LIN {X -173.235,Y +1142.221,Z +0.000,A -20.000,E1 +22.930,E3 +126000.532,E4 +0.000} C_DIS
LIN {X -181.123,Y +1133.734,Z +0.000,A -20.000,E1 +30.868,E3 +126021.288,E4 +0.000} C_DIS
LIN {X -189.654,Y +1120.856,Z +0.000,A -20.000,E1 +39.018,E3 +126043.302,E4 +0.000} C_DIS
LIN {X -195.246,Y +1107.046,Z +0.000,A -20.000,E1 +44.515,E3 +126061.204,E4 +0.000} C_DIS
LIN {X -198.051,Y +1092.368,Z +0.000,A -20.000,E1 +47.947,E3 +126077.730,E4 +0.000} C_DIS
LIN {X -198.143,Y +1081.370,Z +0.000,A -19.806,E1 +49.153,E3 +126089.591,E4 +0.000} C_DIS
LIN {X -197.177,Y +1073.569,Z +0.000,A -17.356,E1 +49.162,E3 +126098.175,E4 +0.000} C_DIS
LIN {X -195.448,Y +1066.139,Z +0.000,A -12.154,E1 +48.512,E3 +126106.770,E4 +0.000} C_DIS
LIN {X -193.346,Y +1058.941,Z +0.000,A -7.133,E1 +47.724,E3 +126115.650,E4 +0.000} C_DIS
LIN {X -191.781,Y +1050.839,Z +0.000,A -3.715,E1 +47.274,E3 +126125.983,E4 +0.000} C_DIS
LIN {X -190.795,Y +1039.355,Z +0.000,A -0.983,E1 +46.842,E3 +126140.643,E4 +0.000} C_DIS
LIN {X -190.395,Y +1028.856,Z +0.000,A -0.089,E1 +46.598,E3 +126154.037,E4 +0.000} C_DIS
LIN {X -190.239,Y +1018.851,Z +0.000,A -0.004,E1 +46.529,E3 +126166.805,E4 +0.000} C_DIS
LIN {X -190.161,Y +1004.975,Z +0.000,A +0.000,E1 +46.506,E3 +126184.519,E4 +0.000} C_DIS
LIN {X -190.142,Y +412.853,Z +0.000,A +0.000,E1 +46.501,E3 +126940.725,E4 +0.000} C_DIS
LIN {X -190.147,Y +401.077,Z +0.000,A +0.000,E1 +46.499,E3 +126955.766,E4 +0.000} C_DIS
LIN {X -190.159,Y +390.929,Z +0.000,A +0.000,E1 +46.494,E3 +126968.732,E4 +0.000} C_DIS
LIN {X -190.174,Y +383.973,Z +0.000,A +0.000,E1 +46.484,E3 +126977.625,E4 +0.000} C_DIS
LIN {X -190.200,Y +373.815,Z +0.000,A +0.000,E1 +46.448,E3 +126990.630,E4 +0.000} C_DIS
LIN {X -190.154,Y +361.003,Z +0.000,A +0.000,E1 +46.303,E3 +127007.124,E4 +0.000} C_DIS
LIN {X -189.772,Y +350.660,Z +0.000,A +0.049,E1 +45.996,E3 +127020.663,E4 +0.000} C_DIS
LIN {X -189.325,Y +346.917,Z +0.000,A +0.243,E1 +45.771,E3 +127025.732,E4 +0.000} C_DIS
LIN {X -188.196,Y +342.754,Z +0.000,A +1.966,E1 +45.249,E3 +127031.740,E4 +0.000} C_DIS
LIN {X -185.199,Y +337.023,Z +0.000,A +6.630,E1 +43.793,E3 +127041.114,E4 +0.000} C_DIS
LIN {X -181.141,Y +331.596,Z +0.000,A +12.274,E1 +41.569,E3 +127051.674,E4 +0.000} C_DIS
LIN {X -176.762,Y +326.804,Z +0.000,A +17.560,E1 +38.898,E3 +127063.098,E4 +0.000} C_DIS
LIN {X -172.184,Y +322.578,Z +0.000,A +19.859,E1 +36.197,E3 +127075.828,E4 +0.000} C_DIS
LIN {X -165.998,Y +317.874,Z +0.000,A +20.000,E1 +32.027,E3 +127095.586,E4 +0.000} C_DIS
LIN {X -160.137,Y +314.334,Z +0.000,A +20.000,E1 +26.368,E3 +127119.955,E4 +0.000} C_DIS
LIN {X -155.624,Y +312.245,Z +0.000,A +20.000,E1 +19.506,E3 +127148.631,E4 +0.000} C_DIS
LIN {X -153.557,Y +311.879,Z +0.000,A +20.000,E1 +11.113,E3 +127184.386,E4 +0.000} C_DIS
LIN {X -155.320,Y +313.348,Z +0.000,A +20.000,E1 +3.401,E3 +127217.570,E4 +0.000} C_DIS
LIN {X -160.005,Y +315.804,Z +0.000,A +20.000,E1 -4.720,E3 +127247.948,E4 +0.000} C_DIS
LIN {X -164.504,Y +318.255,Z +0.000,A +20.000,E1 -10.663,E3 +127267.317,E4 +0.000} C_DIS
LIN {X -170.340,Y +322.684,Z +0.000,A +20.000,E1 -17.457,E3 +127287.349,E4 +0.000} C_DIS
LIN {X -175.568,Y +329.106,Z +0.000,A +20.000,E1 -24.747,E3 +127304.583,E4 +0.000} C_DIS
LIN {X -184.074,Y +340.065,Z +0.000,A +20.000,E1 -33.664,E3 +127327.523,E4 +0.000} C_DIS
LIN {X -190.779,Y +351.388,Z +0.000,A +20.000,E1 -40.083,E3 +127345.301,E4 +0.000} C_DIS
LIN {X -195.254,Y +362.955,Z +0.000,A +20.000,E1 -44.515,E3 +127360.054,E4 +0.000} C_DIS
LIN {X -197.754,Y +374.780,Z +0.000,A +20.000,E1 -47.450,E3 +127373.476,E4 +0.000} C_DIS
LIN {X -198.310,Y +383.215,Z +0.000,A +19.956,E1 -48.698,E3 +127382.600,E4 +0.000} C_DIS
LIN {X -197.912,Y +391.275,Z +0.000,A +18.601,E1 -49.158,E3 +127391.318,E4 +0.000} C_DIS
LIN {X -196.679,Y +398.944,Z +0.000,A +13.989,E1 -48.784,E3 +127399.872,E4 +0.000} C_DIS
LIN {X -194.742,Y +406.288,Z +0.000,A +8.476,E1 -48.001,E3 +127408.555,E4 +0.000} C_DIS
LIN {X -192.748,Y +413.472,Z +0.000,A +3.905,E1 -47.267,E3 +127417.565,E4 +0.000} C_DIS
LIN {X -191.781,Y +419.162,Z +0.000,A +1.739,E1 -46.975,E3 +127424.833,E4 +0.000} C_DIS
LIN {X -190.795,Y +430.646,Z +0.000,A +0.152,E1 -46.707,E3 +127439.494,E4 +0.000} C_DIS
LIN {X -190.395,Y +441.145,Z +0.000,A +0.001,E1 -46.583,E3 +127452.887,E4 +0.000} C_DIS
LIN {X -190.239,Y +451.150,Z +0.000,A -0.000,E1 -46.528,E3 +127465.655,E4 +0.000} C_DIS
LIN {X -190.161,Y +465.026,Z +0.000,A -0.000,E1 -46.506,E3 +127483.370,E4 +0.000} C_DIS
LIN {X -190.142,Y +1057.148,Z +0.000,A -0.000,E1 -46.500,E3 +128239.576,E4 +0.000} C_DIS
LIN {X -190.147,Y +1068.924,Z +0.000,A -0.000,E1 -46.499,E3 +128254.617,E4 +0.000} C_DIS
LIN {X -190.159,Y +1079.072,Z +0.000,A -0.000,E1 -46.493,E3 +128267.582,E4 +0.000} C_DIS
LIN {X -190.174,Y +1086.028,Z +0.000,A -0.000,E1 -46.483,E3 +128276.476,E4 +0.000} C_DIS
LIN {X -190.200,Y +1096.186,Z +0.000,A -0.000,E1 -46.448,E3 +128289.480,E4 +0.000} C_DIS
LIN {X -190.154,Y +1108.998,Z +0.000,A -0.054,E1 -46.295,E3 +128305.975,E4 +0.000} C_DIS
LIN {X -189.772,Y +1119.341,Z +0.000,A -0.752,E1 -45.902,E3 +128319.513,E4 +0.000} C_DIS
LIN {X -189.097,Y +1124.276,Z +0.000,A -2.508,E1 -45.397,E3 +128326.245,E4 +0.000} C_DIS
LIN {X -187.410,Y +1129.069,Z +0.000,A -5.304,E1 -44.585,E3 +128333.418,E4 +0.000} C_DIS
LIN {X -183.899,Y +1134.873,Z +0.000,A -10.372,E1 -42.805,E3 +128343.424,E4 +0.000} C_DIS
LIN {X -179.711,Y +1140.065,Z +0.000,A -15.940,E1 -40.393,E3 +128354.210,E4 +0.000} C_DIS
LIN {X -176.763,Y +1143.197,Z +0.000,A -18.748,E1 -38.674,E3 +128361.948,E4 +0.000} C_DIS
LIN {X -172.185,Y +1147.423,Z +0.000,A -19.971,E1 -36.175,E3 +128374.678,E4 +0.000} C_DIS
LIN {X -165.999,Y +1152.127,Z +0.000,A -20.000,E1 -32.027,E3 +128394.436,E4 +0.000} C_DIS
LIN {X -160.138,Y +1155.667,Z +0.000,A -20.000,E1 -26.368,E3 +128418.806,E4 +0.000} C_DIS
LIN {X -155.625,Y +1157.756,Z +0.000,A -20.000,E1 -19.505,E3 +128447.482,E4 +0.000} C_DIS
LIN {X -153.552,Y +1158.113,Z +0.000,A -20.000,E1 -11.113,E3 +128483.233,E4 +0.000} C_DIS
LIN {X -156.311,Y +1155.540,Z +0.000,A -20.000,E1 -0.839,E3 +128526.593,E4 +0.000} C_DIS
LIN {X -161.281,Y +1151.851,Z +0.000,A -20.000,E1 +7.737,E3 +128556.492,E4 +0.000} C_DIS
LIN {X -167.493,Y +1147.157,Z +0.000,A -20.000,E1 +16.195,E3 +128580.931,E4 +0.000} C_DIS
LIN {X -173.235,Y +1142.221,Z +0.000,A -20.000,E1 +22.930,E3 +128598.233,E4 +0.000} C_DIS
LIN {X -181.123,Y +1133.734,Z +0.000,A -20.000,E1 +30.868,E3 +128618.989,E4 +0.000} C_DIS
LIN {X -189.654,Y +1120.856,Z +0.000,A -20.000,E1 +39.018,E3 +128641.003,E4 +0.000} C_DIS
LIN {X -195.246,Y +1107.046,Z +0.000,A -20.000,E1 +44.515,E3 +128658.905,E4 +0.000} C_DIS
LIN {X -198.051,Y +1092.368,Z +0.000,A -20.000,E1 +47.947,E3 +128675.431,E4 +0.000} C_DIS
LIN {X -198.143,Y +1081.370,Z +0.000,A -19.806,E1 +49.153,E3 +128687.292,E4 +0.000} C_DIS
LIN {X -197.177,Y +1073.569,Z +0.000,A -17.356,E1 +49.162,E3 +128695.876,E4 +0.000} C_DIS
LIN {X -195.448,Y +1066.139,Z +0.000,A -12.154,E1 +48.512,E3 +128704.471,E4 +0.000} C_DIS
LIN {X -193.346,Y +1058.941,Z +0.000,A -7.133,E1 +47.724,E3 +128713.351,E4 +0.000} C_DIS
LIN {X -191.781,Y +1050.839,Z +0.000,A -3.715,E1 +47.274,E3 +128723.684,E4 +0.000} C_DIS
LIN {X -190.795,Y +1039.355,Z +0.000,A -0.983,E1 +46.842,E3 +128738.344,E4 +0.000} C_DIS
LIN {X -190.395,Y +1028.856,Z +0.000,A -0.089,E1 +46.598,E3 +128751.738,E4 +0.000} C_DIS
LIN {X -190.239,Y +1018.851,Z +0.000,A -0.004,E1 +46.529,E3 +128764.506,E4 +0.000} C_DIS
LIN {X -190.161,Y +1004.975,Z +0.000,A +0.000,E1 +46.506,E3 +128782.220,E4 +0.000} C_DIS
LIN {X -190.142,Y +412.853,Z +0.000,A +0.000,E1 +46.501,E3 +129538.426,E4 +0.000} C_DIS
LIN {X -190.147,Y +401.077,Z +0.000,A +0.000,E1 +46.499,E3 +129553.467,E4 +0.000} C_DIS
LIN {X -190.159,Y +390.929,Z +0.000,A +0.000,E1 +46.494,E3 +129566.433,E4 +0.000} C_DIS
LIN {X -190.174,Y +383.973,Z +0.000,A +0.000,E1 +46.484,E3 +129575.326,E4 +0.000} C_DIS
LIN {X -190.200,Y +373.815,Z +0.000,A +0.000,E1 +46.448,E3 +129588.331,E4 +0.000} C_DIS
LIN {X -190.154,Y +361.003,Z +0.000,A +0.000,E1 +46.303,E3 +129604.825,E4 +0.000} C_DIS
LIN {X -189.772,Y +350.660,Z +0.000,A +0.049,E1 +45.996,E3 +129618.364,E4 +0.000} C_DIS
LIN {X -189.325,Y +346.917,Z +0.000,A +0.243,E1 +45.771,E3 +129623.433,E4 +0.000} C_DIS
LIN {X -188.196,Y +342.754,Z +0.000,A +1.966,E1 +45.249,E3 +129629.441,E4 +0.000} C_DIS
LIN {X -185.199,Y +337.023,Z +0.000,A +6.630,E1 +43.793,E3 +129638.815,E4 +0.000} C_DIS
LIN {X -181.141,Y +331.596,Z +0.000,A +12.274,E1 +41.569,E3 +129649.375,E4 +0.000} C_DIS
LIN {X -176.762,Y +326.804,Z +0.000,A +17.560,E1 +38.898,E3 +129660.799,E4 +0.000} C_DIS
LIN {X -172.184,Y +322.578,Z +0.000,A +19.859,E1 +36.197,E3 +129673.529,E4 +0.000} C_DIS
LIN {X -165.998,Y +317.874,Z +0.000,A +20.000,E1 +32.027,E3 +129693.287,E4 +0.000} C_DIS
LIN {X -160.137,Y +314.334,Z +0.000,A +20.000,E1 +26.368,E3 +129717.656,E4 +0.000} C_DIS
LIN {X -155.624,Y +312.245,Z +0.000,A +20.000,E1 +19.506,E3 +129746.332,E4 +0.000} C_DIS
LIN {X -153.557,Y +311.879,Z +0.000,A +20.000,E1 +11.113,E3 +129782.087,E4 +0.000} C_DIS
LIN {X -155.320,Y +313.348,Z +0.000,A +20.000,E1 +3.401,E3 +129815.271,E4 +0.000} C_DIS
LIN {X -160.005,Y +315.804,Z +0.000,A +20.000,E1 -4.720,E3 +129845.649,E4 +0.000} C_DIS
LIN {X -164.504,Y +318.255,Z +0.000,A +20.000,E1 -10.663,E3 +129865.018,E4 +0.000} C_DIS
LIN {X -170.340,Y +322.684,Z +0.000,A +20.000,E1 -17.457,E3 +129885.050,E4 +0.000} C_DIS
LIN {X -175.568,Y +329.106,Z +0.000,A +20.000,E1 -24.747,E3 +129902.284,E4 +0.000} C_DIS
LIN {X -184.074,Y +340.065,Z +0.000,A +20.000,E1 -33.664,E3 +129925.224,E4 +0.000} C_DIS
LIN {X -190.779,Y +351.388,Z +0.000,A +20.000,E1 -40.083,E3 +129943.002,E4 +0.000} C_DIS
LIN {X -195.254,Y +362.955,Z +0.000,A +20.000,E1 -44.515,E3 +129957.755,E4 +0.000} C_DIS
LIN {X -197.754,Y +374.780,Z +0.000,A +20.000,E1 -47.450,E3 +129971.177,E4 +0.000} C_DIS
LIN {X -198.310,Y +383.215,Z +0.000,A +19.956,E1 -48.698,E3 +129980.301,E4 +0.000} C_DIS
LIN {X -197.912,Y +391.275,Z +0.000,A +18.601,E1 -49.158,E3 +129989.019,E4 +0.000} C_DIS
LIN {X -196.679,Y +398.944,Z +0.000,A +13.989,E1 -48.784,E3 +129997.573,E4 +0.000} C_DIS
LIN {X -194.742,Y +406.288,Z +0.000,A +8.476,E1 -48.001,E3 +130006.256,E4 +0.000} C_DIS
LIN {X -192.748,Y +413.472,Z +0.000,A +3.905,E1 -47.267,E3 +130015.266,E4 +0.000} C_DIS
LIN {X -191.781,Y +419.162,Z +0.000,A +1.739,E1 -46.975,E3 +130022.534,E4 +0.000} C_DIS
LIN {X -190.795,Y +430.646,Z +0.000,A +0.152,E1 -46.707,E3 +130037.195,E4 +0.000} C_DIS
LIN {X -190.395,Y +441.145,Z +0.000,A +0.001,E1 -46.583,E3 +130050.588,E4 +0.000} C_DIS
LIN {X -190.239,Y +451.150,Z +0.000,A -0.000,E1 -46.528,E3 +130063.356,E4 +0.000} C_DIS
LIN {X -190.161,Y +465.026,Z +0.000,A -0.000,E1 -46.506,E3 +130081.071,E4 +0.000} C_DIS
LIN {X -190.142,Y +1057.148,Z +0.000,A -0.000,E1 -46.500,E3 +130837.277,E4 +0.000} C_DIS
LIN {X -190.147,Y +1068.924,Z +0.000,A -0.000,E1 -46.499,E3 +130852.318,E4 +0.000} C_DIS
LIN {X -190.159,Y +1079.072,Z +0.000,A -0.000,E1 -46.493,E3 +130865.283,E4 +0.000} C_DIS
LIN {X -190.174,Y +1086.028,Z +0.000,A -0.000,E1 -46.483,E3 +130874.177,E4 +0.000} C_DIS
LIN {X -190.200,Y +1096.186,Z +0.000,A -0.000,E1 -46.448,E3 +130887.181,E4 +0.000} C_DIS
LIN {X -190.154,Y +1108.998,Z +0.000,A -0.054,E1 -46.295,E3 +130903.676,E4 +0.000} C_DIS
LIN {X -189.772,Y +1119.341,Z +0.000,A -0.752,E1 -45.902,E3 +130917.214,E4 +0.000} C_DIS
LIN {X -189.097,Y +1124.276,Z +0.000,A -2.508,E1 -45.397,E3 +130923.946,E4 +0.000} C_DIS
LIN {X -187.410,Y +1129.069,Z +0.000,A -5.304,E1 -44.585,E3 +130931.119,E4 +0.000} C_DIS
LIN {X -183.899,Y +1134.873,Z +0.000,A -10.372,E1 -42.805,E3 +130941.125,E4 +0.000} C_DIS
LIN {X -179.711,Y +1140.065,Z +0.000,A -15.940,E1 -40.393,E3 +130951.911,E4 +0.000} C_DIS
LIN {X -176.763,Y +1143.197,Z +0.000,A -18.748,E1 -38.674,E3 +130959.649,E4 +0.000} C_DIS
LIN {X -172.185,Y +1147.423,Z +0.000,A -19.971,E1 -36.175,E3 +130972.379,E4 +0.000} C_DIS
LIN {X -165.999,Y +1152.127,Z +0.000,A -20.000,E1 -32.027,E3 +130992.137,E4 +0.000} C_DIS
LIN {X -160.138,Y +1155.667,Z +0.000,A -20.000,E1 -26.368,E3 +131016.507,E4 +0.000} C_DIS
LIN {X -155.625,Y +1157.756,Z +0.000,A -20.000,E1 -19.505,E3 +131045.183,E4 +0.000} C_DIS
LIN {X -153.552,Y +1158.113,Z +0.000,A -20.000,E1 -11.113,E3 +131080.934,E4 +0.000} C_DIS
LIN {X -156.311,Y +1155.540,Z +0.000,A -20.000,E1 -0.839,E3 +131124.294,E4 +0.000} C_DIS
LIN {X -161.281,Y +1151.851,Z +0.000,A -20.000,E1 +7.737,E3 +131154.193,E4 +0.000} C_DIS
LIN {X -167.493,Y +1147.157,Z +0.000,A -20.000,E1 +16.195,E3 +131178.632,E4 +0.000} C_DIS
LIN {X -173.235,Y +1142.221,Z +0.000,A -20.000,E1 +22.930,E3 +131195.934,E4 +0.000} C_DIS
LIN {X -181.123,Y +1133.734,Z +0.000,A -20.000,E1 +30.868,E3 +131216.690,E4 +0.000} C_DIS
LIN {X -189.654,Y +1120.856,Z +0.000,A -20.000,E1 +39.018,E3 +131238.704,E4 +0.000} C_DIS
LIN {X -195.246,Y +1107.046,Z +0.000,A -20.000,E1 +44.515,E3 +131256.606,E4 +0.000} C_DIS
LIN {X -198.051,Y +1092.368,Z +0.000,A -20.000,E1 +47.947,E3 +131273.132,E4 +0.000} C_DIS
LIN {X -198.143,Y +1081.370,Z +0.000,A -19.806,E1 +49.153,E3 +131284.993,E4 +0.000} C_DIS
LIN {X -197.177,Y +1073.569,Z +0.000,A -17.356,E1 +49.162,E3 +131293.577,E4 +0.000} C_DIS
LIN {X -195.448,Y +1066.139,Z +0.000,A -12.154,E1 +48.512,E3 +131302.172,E4 +0.000} C_DIS
LIN {X -193.346,Y +1058.941,Z +0.000,A -7.133,E1 +47.724,E3 +131311.052,E4 +0.000} C_DIS
LIN {X -191.781,Y +1050.839,Z +0.000,A -3.715,E1 +47.274,E3 +131321.385,E4 +0.000} C_DIS
LIN {X -190.795,Y +1039.355,Z +0.000,A -0.983,E1 +46.842,E3 +131336.045,E4 +0.000} C_DIS
LIN {X -190.395,Y +1028.856,Z +0.000,A -0.089,E1 +46.598,E3 +131349.439,E4 +0.000} C_DIS
LIN {X -190.239,Y +1018.851,Z +0.000,A -0.004,E1 +46.529,E3 +131362.207,E4 +0.000} C_DIS
LIN {X -190.161,Y +1004.975,Z +0.000,A +0.000,E1 +46.506,E3 +131379.921,E4 +0.000} C_DIS
LIN {X -190.142,Y +412.853,Z +0.000,A +0.000,E1 +46.501,E3 +132136.127,E4 +0.000} C_DIS
LIN {X -190.147,Y +401.077,Z +0.000,A +0.000,E1 +46.499,E3 +132151.168,E4 +0.000} C_DIS
LIN {X -190.159,Y +390.929,Z +0.000,A +0.000,E1 +46.494,E3 +132164.134,E4 +0.000} C_DIS
LIN {X -190.174,Y +383.973,Z +0.000,A +0.000,E1 +46.484,E3 +132173.027,E4 +0.000} C_DIS
LIN {X -190.200,Y +373.815,Z +0.000,A +0.000,E1 +46.448,E3 +132186.032,E4 +0.000} C_DIS
LIN {X -190.154,Y +361.003,Z +0.000,A +0.000,E1 +46.303,E3 +132202.526,E4 +0.000} C_DIS
LIN {X -189.772,Y +350.660,Z +0.000,A +0.049,E1 +45.996,E3 +132216.065,E4 +0.000} C_DIS
LIN {X -189.325,Y +346.917,Z +0.000,A +0.243,E1 +45.771,E3 +132221.134,E4 +0.000} C_DIS
LIN {X -188.196,Y +342.754,Z +0.000,A +1.966,E1 +45.249,E3 +132227.142,E4 +0.000} C_DIS
LIN {X -185.199,Y +337.023,Z +0.000,A +6.630,E1 +43.793,E3 +132236.516,E4 +0.000} C_DIS
LIN {X -181.141,Y +331.596,Z +0.000,A +12.274,E1 +41.569,E3 +132247.076,E4 +0.000} C_DIS
LIN {X -176.762,Y +326.804,Z +0.000,A +17.560,E1 +38.898,E3 +132258.500,E4 +0.000} C_DIS
LIN {X -172.184,Y +322.578,Z +0.000,A +19.859,E1 +36.197,E3 +132271.230,E4 +0.000} C_DIS
LIN {X -165.998,Y +317.874,Z +0.000,A +20.000,E1 +32.027,E3 +132290.988,E4 +0.000} C_DIS
LIN {X -160.137,Y +314.334,Z +0.000,A +20.000,E1 +26.368,E3 +132315.357,E4 +0.000} C_DIS
LIN {X -155.624,Y +312.245,Z +0.000,A +20.000,E1 +19.506,E3 +132344.033,E4 +0.000} C_DIS
LIN {X -153.557,Y +311.879,Z +0.000,A +20.000,E1 +11.113,E3 +132379.788,E4 +0.000} C_DIS
LIN {X -155.320,Y +313.348,Z +0.000,A +20.000,E1 +3.401,E3 +132412.972,E4 +0.000} C_DIS
LIN {X -160.005,Y +315.804,Z +0.000,A +20.000,E1 -4.720,E3 +132443.350,E4 +0.000} C_DIS
LIN {X -164.504,Y +318.255,Z +0.000,A +20.000,E1 -10.663,E3 +132462.719,E4 +0.000} C_DIS
LIN {X -170.340,Y +322.684,Z +0.000,A +20.000,E1 -17.457,E3 +132482.751,E4 +0.000} C_DIS
LIN {X -175.568,Y +329.106,Z +0.000,A +20.000,E1 -24.747,E3 +132499.985,E4 +0.000} C_DIS
LIN {X -184.074,Y +340.065,Z +0.000,A +20.000,E1 -33.664,E3 +132522.925,E4 +0.000} C_DIS
LIN {X -190.779,Y +351.388,Z +0.000,A +20.000,E1 -40.083,E3 +132540.703,E4 +0.000} C_DIS
LIN {X -195.254,Y +362.955,Z +0.000,A +20.000,E1 -44.515,E3 +132555.456,E4 +0.000} C_DIS
LIN {X -197.754,Y +374.780,Z +0.000,A +20.000,E1 -47.450,E3 +132568.878,E4 +0.000} C_DIS
LIN {X -198.310,Y +383.215,Z +0.000,A +19.956,E1 -48.698,E3 +132578.002,E4 +0.000} C_DIS
LIN {X -197.912,Y +391.275,Z +0.000,A +18.601,E1 -49.158,E3 +132586.720,E4 +0.000} C_DIS
LIN {X -196.679,Y +398.944,Z +0.000,A +13.989,E1 -48.784,E3 +132595.274,E4 +0.000} C_DIS
LIN {X -194.742,Y +406.288,Z +0.000,A +8.476,E1 -48.001,E3 +132603.957,E4 +0.000} C_DIS
LIN {X -192.748,Y +413.472,Z +0.000,A +3.905,E1 -47.267,E3 +132612.967,E4 +0.000} C_DIS
LIN {X -191.781,Y +419.162,Z +0.000,A +1.739,E1 -46.975,E3 +132620.235,E4 +0.000} C_DIS
LIN {X -190.795,Y +430.646,Z +0.000,A +0.152,E1 -46.707,E3 +132634.896,E4 +0.000} C_DIS
LIN {X -190.395,Y +441.145,Z +0.000,A +0.001,E1 -46.583,E3 +132648.289,E4 +0.000} C_DIS
LIN {X -190.239,Y +451.150,Z +0.000,A -0.000,E1 -46.528,E3 +132661.057,E4 +0.000} C_DIS
LIN {X -190.161,Y +465.026,Z +0.000,A -0.000,E1 -46.506,E3 +132678.772,E4 +0.000} C_DIS
LIN {X -190.142,Y +1057.148,Z +0.000,A -0.000,E1 -46.500,E3 +133434.978,E4 +0.000} C_DIS
LIN {X -190.147,Y +1068.924,Z +0.000,A -0.000,E1 -46.499,E3 +133450.019,E4 +0.000} C_DIS
LIN {X -190.159,Y +1079.072,Z +0.000,A -0.000,E1 -46.493,E3 +133462.984,E4 +0.000} C_DIS
LIN {X -190.174,Y +1086.028,Z +0.000,A -0.000,E1 -46.483,E3 +133471.878,E4 +0.000} C_DIS
LIN {X -190.200,Y +1096.186,Z +0.000,A -0.000,E1 -46.448,E3 +133484.882,E4 +0.000} C_DIS
LIN {X -190.154,Y +1108.998,Z +0.000,A -0.054,E1 -46.295,E3 +133501.377,E4 +0.000} C_DIS
LIN {X -189.772,Y +1119.341,Z +0.000,A -0.752,E1 -45.902,E3 +133514.915,E4 +0.000} C_DIS
LIN {X -189.097,Y +1124.276,Z +0.000,A -2.508,E1 -45.397,E3 +133521.647,E4 +0.000} C_DIS
LIN {X -187.410,Y +1129.069,Z +0.000,A -5.304,E1 -44.585,E3 +133528.820,E4 +0.000} C_DIS
LIN {X -183.899,Y +1134.873,Z +0.000,A -10.372,E1 -42.805,E3 +133538.826,E4 +0.000} C_DIS
LIN {X -179.711,Y +1140.065,Z +0.000,A -15.940,E1 -40.393,E3 +133549.612,E4 +0.000} C_DIS
LIN {X -176.763,Y +1143.197,Z +0.000,A -18.748,E1 -38.674,E3 +133557.350,E4 +0.000} C_DIS
LIN {X -172.185,Y +1147.423,Z +0.000,A -19.971,E1 -36.175,E3 +133570.080,E4 +0.000} C_DIS
LIN {X -165.999,Y +1152.127,Z +0.000,A -20.000,E1 -32.027,E3 +133589.838,E4 +0.000} C_DIS
LIN {X -160.138,Y +1155.667,Z +0.000,A -20.000,E1 -26.368,E3 +133614.208,E4 +0.000} C_DIS
LIN {X -155.625,Y +1157.756,Z +0.000,A -20.000,E1 -19.505,E3 +133642.884,E4 +0.000} C_DIS
LIN {X -153.552,Y +1158.113,Z +0.000,A -20.000,E1 -11.113,E3 +133678.635,E4 +0.000} C_DIS
LIN {X -156.311,Y +1155.540,Z +0.000,A -20.000,E1 -0.839,E3 +133721.995,E4 +0.000} C_DIS
LIN {X -161.281,Y +1151.851,Z +0.000,A -20.000,E1 +7.737,E3 +133751.894,E4 +0.000} C_DIS
LIN {X -167.493,Y +1147.157,Z +0.000,A -20.000,E1 +16.195,E3 +133776.333,E4 +0.000} C_DIS
LIN {X -173.235,Y +1142.221,Z +0.000,A -20.000,E1 +22.930,E3 +133793.635,E4 +0.000} C_DIS
LIN {X -181.123,Y +1133.734,Z +0.000,A -20.000,E1 +30.868,E3 +133814.391,E4 +0.000} C_DIS
LIN {X -189.654,Y +1120.856,Z +0.000,A -20.000,E1 +39.018,E3 +133836.405,E4 +0.000} C_DIS
LIN {X -195.246,Y +1107.046,Z +0.000,A -20.000,E1 +44.515,E3 +133854.307,E4 +0.000} C_DIS
LIN {X -198.051,Y +1092.368,Z +0.000,A -20.000,E1 +47.947,E3 +133870.833,E4 +0.000} C_DIS
LIN {X -198.143,Y +1081.370,Z +0.000,A -19.806,E1 +49.153,E3 +133882.694,E4 +0.000} C_DIS
LIN {X -197.177,Y +1073.569,Z +0.000,A -17.356,E1 +49.162,E3 +133891.278,E4 +0.000} C_DIS
LIN {X -195.448,Y +1066.139,Z +0.000,A -12.154,E1 +48.512,E3 +133899.873,E4 +0.000} C_DIS
LIN {X -193.346,Y +1058.941,Z +0.000,A -7.133,E1 +47.724,E3 +133908.753,E4 +0.000} C_DIS
LIN {X -191.781,Y +1050.839,Z +0.000,A -3.715,E1 +47.274,E3 +133919.086,E4 +0.000} C_DIS
LIN {X -190.795,Y +1039.355,Z +0.000,A -0.983,E1 +46.842,E3 +133933.746,E4 +0.000} C_DIS
LIN {X -190.395,Y +1028.856,Z +0.000,A -0.089,E1 +46.598,E3 +133947.140,E4 +0.000} C_DIS
LIN {X -190.239,Y +1018.851,Z +0.000,A -0.004,E1 +46.529,E3 +133959.908,E4 +0.000} C_DIS
LIN {X -190.161,Y +1004.975,Z +0.000,A +0.000,E1 +46.506,E3 +133977.622,E4 +0.000} C_DIS
LIN {X -190.142,Y +412.853,Z +0.000,A +0.000,E1 +46.501,E3 +134733.828,E4 +0.000} C_DIS
LIN {X -190.147,Y +401.077,Z +0.000,A +0.000,E1 +46.499,E3 +134748.869,E4 +0.000} C_DIS
LIN {X -190.159,Y +390.929,Z +0.000,A +0.000,E1 +46.494,E3 +134761.835,E4 +0.000} C_DIS
LIN {X -190.174,Y +383.973,Z +0.000,A +0.000,E1 +46.484,E3 +134770.728,E4 +0.000} C_DIS
LIN {X -190.200,Y +373.815,Z +0.000,A +0.000,E1 +46.448,E3 +134783.733,E4 +0.000} C_DIS
LIN {X -190.154,Y +361.003,Z +0.000,A +0.000,E1 +46.303,E3 +134800.227,E4 +0.000} C_DIS
LIN {X -189.772,Y +350.660,Z +0.000,A +0.049,E1 +45.996,E3 +134813.766,E4 +0.000} C_DIS
LIN {X -189.325,Y +346.917,Z +0.000,A +0.243,E1 +45.771,E3 +134818.835,E4 +0.000} C_DIS
LIN {X -188.196,Y +342.754,Z +0.000,A +1.966,E1 +45.249,E3 +134824.843,E4 +0.000} C_DIS
LIN {X -185.199,Y +337.023,Z +0.000,A +6.630,E1 +43.793,E3 +134834.217,E4 +0.000} C_DIS
LIN {X -181.141,Y +331.596,Z +0.000,A +12.274,E1 +41.569,E3 +134844.777,E4 +0.000} C_DIS
LIN {X -176.762,Y +326.804,Z +0.000,A +17.560,E1 +38.898,E3 +134856.201,E4 +0.000} C_DIS
LIN {X -172.184,Y +322.578,Z +0.000,A +19.859,E1 +36.197,E3 +134868.931,E4 +0.000} C_DIS
LIN {X -165.998,Y +317.874,Z +0.000,A +20.000,E1 +32.027,E3 +134888.689,E4 +0.000} C_DIS
LIN {X -160.137,Y +314.334,Z +0.000,A +20.000,E1 +26.368,E3 +134913.058,E4 +0.000} C_DIS
LIN {X -155.624,Y +312.245,Z +0.000,A +20.000,E1 +19.506,E3 +134941.734,E4 +0.000} C_DIS
LIN {X -153.557,Y +311.879,Z +0.000,A +20.000,E1 +11.113,E3 +134977.489,E4 +0.000} C_DIS
LIN {X -155.320,Y +313.348,Z +0.000,A +20.000,E1 +3.401,E3 +135010.673,E4 +0.000} C_DIS
LIN {X -160.005,Y +315.804,Z +0.000,A +20.000,E1 -4.720,E3 +135041.051,E4 +0.000} C_DIS
LIN {X -164.504,Y +318.255,Z +0.000,A +20.000,E1 -10.663,E3 +135060.420,E4 +0.000} C_DIS
LIN {X -170.340,Y +322.684,Z +0.000,A +20.000,E1 -17.457,E3 +135080.452,E4 +0.000} C_DIS
LIN {X -175.568,Y +329.106,Z +0.000,A +20.000,E1 -24.747,E3 +135097.686,E4 +0.000} C_DIS
LIN {X -184.074,Y +340.065,Z +0.000,A +20.000,E1 -33.664,E3 +135120.626,E4 +0.000} C_DIS
LIN {X -190.779,Y +351.388,Z +0.000,A +20.000,E1 -40.083,E3 +135138.404,E4 +0.000} C_DIS
LIN {X -195.254,Y +362.955,Z +0.000,A +20.000,E1 -44.515,E3 +135153.157,E4 +0.000} C_DIS
LIN {X -197.754,Y +374.780,Z +0.000,A +20.000,E1 -47.450,E3 +135166.579,E4 +0.000} C_DIS
LIN {X -198.310,Y +383.215,Z +0.000,A +19.956,E1 -48.698,E3 +135175.703,E4 +0.000} C_DIS
LIN {X -197.912,Y +391.275,Z +0.000,A +18.601,E1 -49.158,E3 +135184.421,E4 +0.000} C_DIS
LIN {X -196.679,Y +398.944,Z +0.000,A +13.989,E1 -48.784,E3 +135192.975,E4 +0.000} C_DIS
LIN {X -194.742,Y +406.288,Z +0.000,A +8.476,E1 -48.001,E3 +135201.658,E4 +0.000} C_DIS
LIN {X -192.748,Y +413.472,Z +0.000,A +3.905,E1 -47.267,E3 +135210.668,E4 +0.000} C_DIS
LIN {X -191.781,Y +419.162,Z +0.000,A +1.739,E1 -46.975,E3 +135217.936,E4 +0.000} C_DIS
LIN {X -190.795,Y +430.646,Z +0.000,A +0.152,E1 -46.707,E3 +135232.597,E4 +0.000} C_DIS
LIN {X -190.395,Y +441.145,Z +0.000,A +0.001,E1 -46.583,E3 +135245.990,E4 +0.000} C_DIS
LIN {X -190.239,Y +451.150,Z +0.000,A -0.000,E1 -46.528,E3 +135258.758,E4 +0.000} C_DIS
LIN {X -190.161,Y +465.026,Z +0.000,A -0.000,E1 -46.506,E3 +135276.473,E4 +0.000} C_DIS
LIN {X -190.142,Y +1057.148,Z +0.000,A -0.000,E1 -46.500,E3 +136032.679,E4 +0.000} C_DIS
LIN {X -190.147,Y +1068.924,Z +0.000,A -0.000,E1 -46.499,E3 +136047.720,E4 +0.000} C_DIS
LIN {X -190.159,Y +1079.072,Z +0.000,A -0.000,E1 -46.493,E3 +136060.685,E4 +0.000} C_DIS
LIN {X -190.174,Y +1086.028,Z +0.000,A -0.000,E1 -46.483,E3 +136069.579,E4 +0.000} C_DIS
LIN {X -190.200,Y +1096.186,Z +0.000,A -0.000,E1 -46.448,E3 +136082.583,E4 +0.000} C_DIS
LIN {X -190.154,Y +1108.998,Z +0.000,A -0.054,E1 -46.295,E3 +136099.078,E4 +0.000} C_DIS
LIN {X -189.772,Y +1119.341,Z +0.000,A -0.752,E1 -45.902,E3 +136112.616,E4 +0.000} C_DIS
LIN {X -189.097,Y +1124.276,Z +0.000,A -2.508,E1 -45.397,E3 +136119.348,E4 +0.000} C_DIS
LIN {X -187.410,Y +1129.069,Z +0.000,A -5.304,E1 -44.585,E3 +136126.521,E4 +0.000} C_DIS
LIN {X -183.899,Y +1134.873,Z +0.000,A -10.372,E1 -42.805,E3 +136136.527,E4 +0.000} C_DIS
LIN {X -179.711,Y +1140.065,Z +0.000,A -15.940,E1 -40.393,E3 +136147.313,E4 +0.000} C_DIS
LIN {X -176.763,Y +1143.197,Z +0.000,A -18.748,E1 -38.674,E3 +136155.051,E4 +0.000} C_DIS
LIN {X -172.185,Y +1147.423,Z +0.000,A -19.971,E1 -36.175,E3 +136167.781,E4 +0.000} C_DIS
LIN {X -165.999,Y +1152.127,Z +0.000,A -20.000,E1 -32.027,E3 +136187.539,E4 +0.000} C_DIS
LIN {X -160.138,Y +1155.667,Z +0.000,A -20.000,E1 -26.368,E3 +136211.909,E4 +0.000} C_DIS
LIN {X -155.625,Y +1157.756,Z +0.000,A -20.000,E1 -19.505,E3 +136240.585,E4 +0.000} C_DIS
LIN {X -153.552,Y +1158.113,Z +0.000,A -20.000,E1 -11.113,E3 +136276.336,E4 +0.000} C_DIS
LIN {X -156.311,Y +1155.540,Z +0.000,A -20.000,E1 -0.839,E3 +136319.696,E4 +0.000} C_DIS
LIN {X -161.281,Y +1151.851,Z +0.000,A -20.000,E1 +7.737,E3 +136349.595,E4 +0.000} C_DIS
LIN {X -167.493,Y +1147.157,Z +0.000,A -20.000,E1 +16.195,E3 +136374.034,E4 +0.000} C_DIS
LIN {X -173.235,Y +1142.221,Z +0.000,A -20.000,E1 +22.930,E3 +136391.336,E4 +0.000} C_DIS
LIN {X -181.123,Y +1133.734,Z +0.000,A -20.000,E1 +30.868,E3 +136412.092,E4 +0.000} C_DIS
LIN {X -189.654,Y +1120.856,Z +0.000,A -20.000,E1 +39.018,E3 +136434.106,E4 +0.000} C_DIS
LIN {X -195.246,Y +1107.046,Z +0.000,A -20.000,E1 +44.515,E3 +136452.008,E4 +0.000} C_DIS
LIN {X -198.051,Y +1092.368,Z +0.000,A -20.000,E1 +47.947,E3 +136468.534,E4 +0.000} C_DIS
LIN {X -198.143,Y +1081.370,Z +0.000,A -19.806,E1 +49.153,E3 +136480.395,E4 +0.000} C_DIS
LIN {X -197.177,Y +1073.569,Z +0.000,A -17.356,E1 +49.162,E3 +136488.979,E4 +0.000} C_DIS
LIN {X -195.448,Y +1066.139,Z +0.000,A -12.154,E1 +48.512,E3 +136497.574,E4 +0.000} C_DIS
LIN {X -193.346,Y +1058.941,Z +0.000,A -7.133,E1 +47.724,E3 +136506.454,E4 +0.000} C_DIS
LIN {X -191.781,Y +1050.839,Z +0.000,A -3.715,E1 +47.274,E3 +136516.787,E4 +0.000} C_DIS
LIN {X -190.795,Y +1039.355,Z +0.000,A -0.983,E1 +46.842,E3 +136531.447,E4 +0.000} C_DIS
LIN {X -190.395,Y +1028.856,Z +0.000,A -0.089,E1 +46.598,E3 +136544.841,E4 +0.000} C_DIS
LIN {X -190.239,Y +1018.851,Z +0.000,A -0.004,E1 +46.529,E3 +136557.609,E4 +0.000} C_DIS
LIN {X -190.161,Y +1004.975,Z +0.000,A +0.000,E1 +46.506,E3 +136575.323,E4 +0.000} C_DIS
LIN {X -190.142,Y +412.853,Z +0.000,A +0.000,E1 +46.501,E3 +137331.529,E4 +0.000} C_DIS
LIN {X -190.147,Y +401.077,Z +0.000,A +0.000,E1 +46.499,E3 +137346.570,E4 +0.000} C_DIS
LIN {X -190.159,Y +390.929,Z +0.000,A +0.000,E1 +46.494,E3 +137359.536,E4 +0.000} C_DIS
LIN {X -190.174,Y +383.973,Z +0.000,A +0.000,E1 +46.484,E3 +137368.429,E4 +0.000} C_DIS
LIN {X -190.200,Y +373.815,Z +0.000,A +0.000,E1 +46.448,E3 +137381.434,E4 +0.000} C_DIS
LIN {X -190.154,Y +361.003,Z +0.000,A +0.000,E1 +46.303,E3 +137397.928,E4 +0.000} C_DIS
LIN {X -189.772,Y +350.660,Z +0.000,A +0.049,E1 +45.996,E3 +137411.467,E4 +0.000} C_DIS
LIN {X -189.325,Y +346.917,Z +0.000,A +0.243,E1 +45.771,E3 +137416.536,E4 +0.000} C_DIS
LIN {X -188.196,Y +342.754,Z +0.000,A +1.966,E1 +45.249,E3 +137422.544,E4 +0.000} C_DIS
LIN {X -185.199,Y +337.023,Z +0.000,A +6.630,E1 +43.793,E3 +137431.918,E4 +0.000} C_DIS
LIN {X -181.141,Y +331.596,Z +0.000,A +12.274,E1 +41.569,E3 +137442.478,E4 +0.000} C_DIS
LIN {X -176.762,Y +326.804,Z +0.000,A +17.560,E1 +38.898,E3 +137453.902,E4 +0.000} C_DIS
LIN {X -172.184,Y +322.578,Z +0.000,A +19.859,E1 +36.197,E3 +137466.632,E4 +0.000} C_DIS
LIN {X -165.998,Y +317.874,Z +0.000,A +20.000,E1 +32.027,E3 +137486.390,E4 +0.000} C_DIS
LIN {X -160.137,Y +314.334,Z +0.000,A +20.000,E1 +26.368,E3 +137510.759,E4 +0.000} C_DIS
LIN {X -155.624,Y +312.245,Z +0.000,A +20.000,E1 +19.506,E3 +137539.435,E4 +0.000} C_DIS
LIN {X -153.557,Y +311.879,Z +0.000,A +20.000,E1 +11.113,E3 +137575.190,E4 +0.000} C_DIS
LIN {X -155.320,Y +313.348,Z +0.000,A +20.000,E1 +3.401,E3 +137608.374,E4 +0.000} C_DIS
LIN {X -160.005,Y +315.804,Z +0.000,A +20.000,E1 -4.720,E3 +137638.752,E4 +0.000} C_DIS
LIN {X -164.504,Y +318.255,Z +0.000,A +20.000,E1 -10.663,E3 +137658.121,E4 +0.000} C_DIS
LIN {X -170.340,Y +322.684,Z +0.000,A +20.000,E1 -17.457,E3 +137678.153,E4 +0.000} C_DIS
LIN {X -175.568,Y +329.106,Z +0.000,A +20.000,E1 -24.747,E3 +137695.387,E4 +0.000} C_DIS
LIN {X -184.074,Y +340.065,Z +0.000,A +20.000,E1 -33.664,E3 +137718.327,E4 +0.000} C_DIS
LIN {X -190.779,Y +351.388,Z +0.000,A +20.000,E1 -40.083,E3 +137736.105,E4 +0.000} C_DIS
LIN {X -195.254,Y +362.955,Z +0.000,A +20.000,E1 -44.515,E3 +137750.858,E4 +0.000} C_DIS
LIN {X -197.754,Y +374.780,Z +0.000,A +20.000,E1 -47.450,E3 +137764.280,E4 +0.000} C_DIS
LIN {X -198.310,Y +383.215,Z +0.000,A +19.956,E1 -48.698,E3 +137773.404,E4 +0.000} C_DIS
LIN {X -197.912,Y +391.275,Z +0.000,A +18.601,E1 -49.158,E3 +137782.122,E4 +0.000} C_DIS
LIN {X -196.679,Y +398.944,Z +0.000,A +13.989,E1 -48.784,E3 +137790.676,E4 +0.000} C_DIS
LIN {X -194.742,Y +406.288,Z +0.000,A +8.476,E1 -48.001,E3 +137799.359,E4 +0.000} C_DIS
LIN {X -192.748,Y +413.472,Z +0.000,A +3.905,E1 -47.267,E3 +137808.369,E4 +0.000} C_DIS
LIN {X -191.781,Y +419.162,Z +0.000,A +1.739,E1 -46.975,E3 +137815.637,E4 +0.000} C_DIS
LIN {X -190.795,Y +430.646,Z +0.000,A +0.152,E1 -46.707,E3 +137830.298,E4 +0.000} C_DIS
LIN {X -190.395,Y +441.145,Z +0.000,A +0.001,E1 -46.583,E3 +137843.691,E4 +0.000} C_DIS
LIN {X -190.239,Y +451.150,Z +0.000,A -0.000,E1 -46.528,E3 +137856.459,E4 +0.000} C_DIS
LIN {X -190.161,Y +465.026,Z +0.000,A -0.000,E1 -46.506,E3 +137874.174,E4 +0.000} C_DIS
LIN {X -190.142,Y +1057.148,Z +0.000,A -0.000,E1 -46.500,E3 +138630.380,E4 +0.000} C_DIS
LIN {X -190.147,Y +1068.924,Z +0.000,A -0.000,E1 -46.499,E3 +138645.421,E4 +0.000} C_DIS
LIN {X -190.159,Y +1079.072,Z +0.000,A -0.000,E1 -46.493,E3 +138658.386,E4 +0.000} C_DIS
LIN {X -190.174,Y +1086.028,Z +0.000,A -0.000,E1 -46.483,E3 +138667.280,E4 +0.000} C_DIS
LIN {X -190.200,Y +1096.186,Z +0.000,A -0.000,E1 -46.448,E3 +138680.284,E4 +0.000} C_DIS
LIN {X -190.154,Y +1108.998,Z +0.000,A -0.054,E1 -46.295,E3 +138696.779,E4 +0.000} C_DIS
LIN {X -189.772,Y +1119.341,Z +0.000,A -0.752,E1 -45.902,E3 +138710.317,E4 +0.000} C_DIS
LIN {X -189.097,Y +1124.276,Z +0.000,A -2.508,E1 -45.397,E3 +138717.049,E4 +0.000} C_DIS
LIN {X -187.410,Y +1129.069,Z +0.000,A -5.304,E1 -44.585,E3 +138724.222,E4 +0.000} C_DIS
LIN {X -183.899,Y +1134.873,Z +0.000,A -10.372,E1 -42.805,E3 +138734.228,E4 +0.000} C_DIS
LIN {X -179.711,Y +1140.065,Z +0.000,A -15.940,E1 -40.393,E3 +138745.014,E4 +0.000} C_DIS
LIN {X -176.763,Y +1143.197,Z +0.000,A -18.748,E1 -38.674,E3 +138752.752,E4 +0.000} C_DIS
LIN {X -172.185,Y +1147.423,Z +0.000,A -19.971,E1 -36.175,E3 +138765.482,E4 +0.000} C_DIS
LIN {X -165.999,Y +1152.127,Z +0.000,A -20.000,E1 -32.027,E3 +138785.240,E4 +0.000} C_DIS
LIN {X -160.138,Y +1155.667,Z +0.000,A -20.000,E1 -26.368,E3 +138809.610,E4 +0.000} C_DIS
LIN {X -155.625,Y +1157.756,Z +0.000,A -20.000,E1 -19.505,E3 +138838.286,E4 +0.000} C_DIS
LIN {X -153.552,Y +1158.113,Z +0.000,A -20.000,E1 -11.113,E3 +138874.037,E4 +0.000} C_DIS
LIN {X -156.311,Y +1155.540,Z +0.000,A -20.000,E1 -0.839,E3 +138917.397,E4 +0.000} C_DIS
LIN {X -161.281,Y +1151.851,Z +0.000,A -20.000,E1 +7.737,E3 +138947.296,E4 +0.000} C_DIS
LIN {X -167.493,Y +1147.157,Z +0.000,A -20.000,E1 +16.195,E3 +138971.735,E4 +0.000} C_DIS
LIN {X -173.235,Y +1142.221,Z +0.000,A -20.000,E1 +22.930,E3 +138989.037,E4 +0.000} C_DIS
LIN {X -181.123,Y +1133.734,Z +0.000,A -20.000,E1 +30.868,E3 +139009.793,E4 +0.000} C_DIS
LIN {X -189.654,Y +1120.856,Z +0.000,A -20.000,E1 +39.018,E3 +139031.807,E4 +0.000} C_DIS
LIN {X -195.246,Y +1107.046,Z +0.000,A -20.000,E1 +44.515,E3 +139049.709,E4 +0.000} C_DIS
LIN {X -198.051,Y +1092.368,Z +0.000,A -20.000,E1 +47.947,E3 +139066.235,E4 +0.000} C_DIS
LIN {X -198.143,Y +1081.370,Z +0.000,A -19.806,E1 +49.153,E3 +139078.096,E4 +0.000} C_DIS
LIN {X -197.177,Y +1073.569,Z +0.000,A -17.356,E1 +49.162,E3 +139086.680,E4 +0.000} C_DIS
LIN {X -195.448,Y +1066.139,Z +0.000,A -12.154,E1 +48.512,E3 +139095.275,E4 +0.000} C_DIS
LIN {X -193.346,Y +1058.941,Z +0.000,A -7.133,E1 +47.724,E3 +139104.155,E4 +0.000} C_DIS
LIN {X -191.781,Y +1050.839,Z +0.000,A -3.715,E1 +47.274,E3 +139114.488,E4 +0.000} C_DIS
LIN {X -190.795,Y +1039.355,Z +0.000,A -0.983,E1 +46.842,E3 +139129.148,E4 +0.000} C_DIS
LIN {X -190.395,Y +1028.856,Z +0.000,A -0.089,E1 +46.598,E3 +139142.542,E4 +0.000} C_DIS
LIN {X -190.239,Y +1018.851,Z +0.000,A -0.004,E1 +46.529,E3 +139155.310,E4 +0.000} C_DIS
LIN {X -190.161,Y +1004.975,Z +0.000,A +0.000,E1 +46.506,E3 +139173.024,E4 +0.000} C_DIS
LIN {X -190.142,Y +412.853,Z +0.000,A +0.000,E1 +46.501,E3 +139929.230,E4 +0.000} C_DIS
LIN {X -190.147,Y +401.077,Z +0.000,A +0.000,E1 +46.499,E3 +139944.271,E4 +0.000} C_DIS
LIN {X -190.159,Y +390.929,Z +0.000,A +0.000,E1 +46.494,E3 +139957.237,E4 +0.000} C_DIS
LIN {X -190.174,Y +383.973,Z +0.000,A +0.000,E1 +46.484,E3 +139966.130,E4 +0.000} C_DIS
LIN {X -190.200,Y +373.815,Z +0.000,A +0.000,E1 +46.448,E3 +139979.135,E4 +0.000} C_DIS
LIN {X -190.154,Y +361.003,Z +0.000,A +0.000,E1 +46.303,E3 +139995.629,E4 +0.000} C_DIS
LIN {X -189.772,Y +350.660,Z +0.000,A +0.049,E1 +45.996,E3 +140009.168,E4 +0.000} C_DIS
LIN {X -189.325,Y +346.917,Z +0.000,A +0.243,E1 +45.771,E3 +140014.237,E4 +0.000} C_DIS
LIN {X -188.196,Y +342.754,Z +0.000,A +1.966,E1 +45.249,E3 +140020.245,E4 +0.000} C_DIS
LIN {X -185.199,Y +337.023,Z +0.000,A +6.630,E1 +43.793,E3 +140029.619,E4 +0.000} C_DIS
LIN {X -181.141,Y +331.596,Z +0.000,A +12.274,E1 +41.569,E3 +140040.179,E4 +0.000} C_DIS
LIN {X -176.762,Y +326.804,Z +0.000,A +17.560,E1 +38.898,E3 +140051.603,E4 +0.000} C_DIS
LIN {X -172.184,Y +322.578,Z +0.000,A +19.859,E1 +36.197,E3 +140064.333,E4 +0.000} C_DIS
LIN {X -165.998,Y +317.874,Z +0.000,A +20.000,E1 +32.027,E3 +140084.091,E4 +0.000} C_DIS
LIN {X -160.137,Y +314.334,Z +0.000,A +20.000,E1 +26.368,E3 +140108.460,E4 +0.000} C_DIS
LIN {X -155.624,Y +312.245,Z +0.000,A +20.000,E1 +19.506,E3 +140137.136,E4 +0.000} C_DIS
LIN {X -153.557,Y +311.879,Z +0.000,A +20.000,E1 +11.113,E3 +140172.891,E4 +0.000} C_DIS
LIN {X -155.320,Y +313.348,Z +0.000,A +20.000,E1 +3.401,E3 +140206.075,E4 +0.000} C_DIS
LIN {X -160.005,Y +315.804,Z +0.000,A +20.000,E1 -4.720,E3 +140236.453,E4 +0.000} C_DIS
LIN {X -164.504,Y +318.255,Z +0.000,A +20.000,E1 -10.663,E3 +140255.822,E4 +0.000} C_DIS
LIN {X -170.340,Y +322.684,Z +0.000,A +20.000,E1 -17.457,E3 +140275.854,E4 +0.000} C_DIS
LIN {X -175.568,Y +329.106,Z +0.000,A +20.000,E1 -24.747,E3 +140293.088,E4 +0.000} C_DIS
LIN {X -184.074,Y +340.065,Z +0.000,A +20.000,E1 -33.664,E3 +140316.028,E4 +0.000} C_DIS
LIN {X -190.779,Y +351.388,Z +0.000,A +20.000,E1 -40.083,E3 +140333.806,E4 +0.000} C_DIS
LIN {X -195.254,Y +362.955,Z +0.000,A +20.000,E1 -44.515,E3 +140348.559,E4 +0.000} C_DIS
LIN {X -197.754,Y +374.780,Z +0.000,A +20.000,E1 -47.450,E3 +140361.981,E4 +0.000} C_DIS
LIN {X -198.310,Y +383.215,Z +0.000,A +19.956,E1 -48.698,E3 +140371.105,E4 +0.000} C_DIS
LIN {X -197.912,Y +391.275,Z +0.000,A +18.601,E1 -49.158,E3 +140379.823,E4 +0.000} C_DIS
LIN {X -196.679,Y +398.944,Z +0.000,A +13.989,E1 -48.784,E3 +140388.377,E4 +0.000} C_DIS
LIN {X -194.742,Y +406.288,Z +0.000,A +8.476,E1 -48.001,E3 +140397.060,E4 +0.000} C_DIS
LIN {X -192.748,Y +413.472,Z +0.000,A +3.905,E1 -47.267,E3 +140406.070,E4 +0.000} C_DIS
LIN {X -191.781,Y +419.162,Z +0.000,A +1.739,E1 -46.975,E3 +140413.338,E4 +0.000} C_DIS
LIN {X -190.795,Y +430.646,Z +0.000,A +0.152,E1 -46.707,E3 +140427.999,E4 +0.000} C_DIS
LIN {X -190.395,Y +441.145,Z +0.000,A +0.001,E1 -46.583,E3 +140441.392,E4 +0.000} C_DIS
LIN {X -190.239,Y +451.150,Z +0.000,A -0.000,E1 -46.528,E3 +140454.160,E4 +0.000} C_DIS
LIN {X -190.161,Y +465.026,Z +0.000,A -0.000,E1 -46.506,E3 +140471.875,E4 +0.000} C_DIS
LIN {X -190.142,Y +1057.148,Z +0.000,A -0.000,E1 -46.500,E3 +141228.081,E4 +0.000} C_DIS
LIN {X -190.147,Y +1068.924,Z +0.000,A -0.000,E1 -46.499,E3 +141243.122,E4 +0.000} C_DIS
LIN {X -190.159,Y +1079.072,Z +0.000,A -0.000,E1 -46.493,E3 +141256.087,E4 +0.000} C_DIS
LIN {X -190.174,Y +1086.028,Z +0.000,A -0.000,E1 -46.483,E3 +141264.981,E4 +0.000} C_DIS
LIN {X -190.200,Y +1096.186,Z +0.000,A -0.000,E1 -46.448,E3 +141277.985,E4 +0.000} C_DIS
LIN {X -190.154,Y +1108.998,Z +0.000,A -0.054,E1 -46.295,E3 +141294.480,E4 +0.000} C_DIS
LIN {X -189.772,Y +1119.341,Z +0.000,A -0.752,E1 -45.902,E3 +141308.018,E4 +0.000} C_DIS
LIN {X -189.097,Y +1124.276,Z +0.000,A -2.508,E1 -45.397,E3 +141314.750,E4 +0.000} C_DIS
LIN {X -187.410,Y +1129.069,Z +0.000,A -5.304,E1 -44.585,E3 +141321.923,E4 +0.000} C_DIS
LIN {X -183.899,Y +1134.873,Z +0.000,A -10.372,E1 -42.805,E3 +141331.929,E4 +0.000} C_DIS
LIN {X -179.711,Y +1140.065,Z +0.000,A -15.940,E1 -40.393,E3 +141342.715,E4 +0.000} C_DIS
LIN {X -176.763,Y +1143.197,Z +0.000,A -18.748,E1 -38.674,E3 +141350.453,E4 +0.000} C_DIS
LIN {X -172.185,Y +1147.423,Z +0.000,A -19.971,E1 -36.175,E3 +141363.183,E4 +0.000} C_DIS
LIN {X -165.999,Y +1152.127,Z +0.000,A -20.000,E1 -32.027,E3 +141382.941,E4 +0.000} C_DIS
LIN {X -160.138,Y +1155.667,Z +0.000,A -20.000,E1 -26.368,E3 +141407.311,E4 +0.000} C_DIS
LIN {X -155.625,Y +1157.756,Z +0.000,A -20.000,E1 -19.505,E3 +141435.987,E4 +0.000} C_DIS
LIN {X -153.552,Y +1158.113,Z +0.000,A -20.000,E1 -11.113,E3 +141471.738,E4 +0.000} C_DIS
LIN {X -156.311,Y +1155.540,Z +0.000,A -20.000,E1 -0.839,E3 +141515.098,E4 +0.000} C_DIS
LIN {X -161.281,Y +1151.851,Z +0.000,A -20.000,E1 +7.737,E3 +141544.997,E4 +0.000} C_DIS
LIN {X -167.493,Y +1147.157,Z +0.000,A -20.000,E1 +16.195,E3 +141569.436,E4 +0.000} C_DIS
LIN {X -173.235,Y +1142.221,Z +0.000,A -20.000,E1 +22.930,E3 +141586.738,E4 +0.000} C_DIS
LIN {X -181.123,Y +1133.734,Z +0.000,A -20.000,E1 +30.868,E3 +141607.494,E4 +0.000} C_DIS
LIN {X -189.654,Y +1120.856,Z +0.000,A -20.000,E1 +39.018,E3 +141629.508,E4 +0.000} C_DIS
LIN {X -195.246,Y +1107.046,Z +0.000,A -20.000,E1 +44.515,E3 +141647.410,E4 +0.000} C_DIS
LIN {X -198.051,Y +1092.368,Z +0.000,A -20.000,E1 +47.947,E3 +141663.936,E4 +0.000} C_DIS
LIN {X -198.143,Y +1081.370,Z +0.000,A -19.806,E1 +49.153,E3 +141675.797,E4 +0.000} C_DIS
LIN {X -197.177,Y +1073.569,Z +0.000,A -17.356,E1 +49.162,E3 +141684.381,E4 +0.000} C_DIS
LIN {X -195.448,Y +1066.139,Z +0.000,A -12.154,E1 +48.512,E3 +141692.976,E4 +0.000} C_DIS
LIN {X -193.346,Y +1058.941,Z +0.000,A -7.133,E1 +47.724,E3 +141701.856,E4 +0.000} C_DIS
LIN {X -191.781,Y +1050.839,Z +0.000,A -3.715,E1 +47.274,E3 +141712.189,E4 +0.000} C_DIS
LIN {X -190.795,Y +1039.355,Z +0.000,A -0.983,E1 +46.842,E3 +141726.849,E4 +0.000} C_DIS
LIN {X -190.395,Y +1028.856,Z +0.000,A -0.089,E1 +46.598,E3 +141740.243,E4 +0.000} C_DIS
LIN {X -190.239,Y +1018.851,Z +0.000,A -0.004,E1 +46.529,E3 +141753.011,E4 +0.000} C_DIS
LIN {X -190.161,Y +1004.975,Z +0.000,A +0.000,E1 +46.506,E3 +141770.725,E4 +0.000} C_DIS
LIN {X -190.142,Y +412.853,Z +0.000,A +0.000,E1 +46.501,E3 +142526.931,E4 +0.000} C_DIS
LIN {X -190.147,Y +401.077,Z +0.000,A +0.000,E1 +46.499,E3 +142541.972,E4 +0.000} C_DIS
LIN {X -190.159,Y +390.929,Z +0.000,A +0.000,E1 +46.494,E3 +142554.938,E4 +0.000} C_DIS
LIN {X -190.174,Y +383.973,Z +0.000,A +0.000,E1 +46.484,E3 +142563.831,E4 +0.000} C_DIS
LIN {X -190.200,Y +373.815,Z +0.000,A +0.000,E1 +46.448,E3 +142576.836,E4 +0.000} C_DIS
LIN {X -190.154,Y +361.003,Z +0.000,A +0.000,E1 +46.303,E3 +142593.330,E4 +0.000} C_DIS
LIN {X -189.772,Y +350.660,Z +0.000,A +0.049,E1 +45.996,E3 +142606.869,E4 +0.000} C_DIS
LIN {X -189.325,Y +346.917,Z +0.000,A +0.243,E1 +45.771,E3 +142611.938,E4 +0.000} C_DIS
LIN {X -188.196,Y +342.754,Z +0.000,A +1.966,E1 +45.249,E3 +142617.946,E4 +0.000} C_DIS
LIN {X -185.199,Y +337.023,Z +0.000,A +6.630,E1 +43.793,E3 +142627.320,E4 +0.000} C_DIS
LIN {X -181.141,Y +331.596,Z +0.000,A +12.274,E1 +41.569,E3 +142637.880,E4 +0.000} C_DIS
LIN {X -176.762,Y +326.804,Z +0.000,A +17.560,E1 +38.898,E3 +142649.304,E4 +0.000} C_DIS
LIN {X -172.184,Y +322.578,Z +0.000,A +19.859,E1 +36.197,E3 +142662.034,E4 +0.000} C_DIS
LIN {X -165.998,Y +317.874,Z +0.000,A +20.000,E1 +32.027,E3 +142681.792,E4 +0.000} C_DIS
LIN {X -160.137,Y +314.334,Z +0.000,A +20.000,E1 +26.368,E3 +142706.161,E4 +0.000} C_DIS
LIN {X -155.624,Y +312.245,Z +0.000,A +20.000,E1 +19.506,E3 +142734.837,E4 +0.000} C_DIS
LIN {X -153.557,Y +311.879,Z +0.000,A +20.000,E1 +11.113,E3 +142770.592,E4 +0.000} C_DIS
LIN {X -155.320,Y +313.348,Z +0.000,A +20.000,E1 +3.401,E3 +142803.776,E4 +0.000} C_DIS
LIN {X -160.005,Y +315.804,Z +0.000,A +20.000,E1 -4.720,E3 +142834.154,E4 +0.000} C_DIS
LIN {X -164.504,Y +318.255,Z +0.000,A +20.000,E1 -10.663,E3 +142853.523,E4 +0.000} C_DIS
LIN {X -170.340,Y +322.684,Z +0.000,A +20.000,E1 -17.457,E3 +142873.555,E4 +0.000} C_DIS
LIN {X -175.568,Y +329.106,Z +0.000,A +20.000,E1 -24.747,E3 +142890.789,E4 +0.000} C_DIS
LIN {X -184.074,Y +340.065,Z +0.000,A +20.000,E1 -33.664,E3 +142913.729,E4 +0.000} C_DIS
LIN {X -190.779,Y +351.388,Z +0.000,A +20.000,E1 -40.083,E3 +142931.507,E4 +0.000} C_DIS
LIN {X -195.254,Y +362.955,Z +0.000,A +20.000,E1 -44.515,E3 +142946.260,E4 +0.000} C_DIS
LIN {X -197.754,Y +374.780,Z +0.000,A +20.000,E1 -47.450,E3 +142959.682,E4 +0.000} C_DIS
LIN {X -198.310,Y +383.215,Z +0.000,A +19.956,E1 -48.698,E3 +142968.806,E4 +0.000} C_DIS
LIN {X -197.912,Y +391.275,Z +0.000,A +18.601,E1 -49.158,E3 +142977.524,E4 +0.000} C_DIS
LIN {X -196.679,Y +398.944,Z +0.000,A +13.989,E1 -48.784,E3 +142986.078,E4 +0.000} C_DIS
LIN {X -194.742,Y +406.288,Z +0.000,A +8.476,E1 -48.001,E3 +142994.761,E4 +0.000} C_DIS
LIN {X -192.748,Y +413.472,Z +0.000,A +3.905,E1 -47.267,E3 +143003.771,E4 +0.000} C_DIS
LIN {X -191.781,Y +419.162,Z +0.000,A +1.739,E1 -46.975,E3 +143011.039,E4 +0.000} C_DIS
LIN {X -190.795,Y +430.646,Z +0.000,A +0.152,E1 -46.707,E3 +143025.700,E4 +0.000} C_DIS
LIN {X -190.395,Y +441.145,Z +0.000,A +0.001,E1 -46.583,E3 +143039.093,E4 +0.000} C_DIS
LIN {X -190.239,Y +451.150,Z +0.000,A -0.000,E1 -46.528,E3 +143051.861,E4 +0.000} C_DIS
LIN {X -190.161,Y +465.026,Z +0.000,A -0.000,E1 -46.506,E3 +143069.576,E4 +0.000} C_DIS
LIN {X -190.142,Y +1057.148,Z +0.000,A -0.000,E1 -46.500,E3 +143825.782,E4 +0.000} C_DIS
LIN {X -190.147,Y +1068.924,Z +0.000,A -0.000,E1 -46.499,E3 +143840.823,E4 +0.000} C_DIS
LIN {X -190.159,Y +1079.072,Z +0.000,A -0.000,E1 -46.493,E3 +143853.788,E4 +0.000} C_DIS
LIN {X -190.174,Y +1086.028,Z +0.000,A -0.000,E1 -46.483,E3 +143862.682,E4 +0.000} C_DIS
LIN {X -190.200,Y +1096.186,Z +0.000,A -0.000,E1 -46.448,E3 +143875.686,E4 +0.000} C_DIS
LIN {X -190.154,Y +1108.998,Z +0.000,A -0.054,E1 -46.295,E3 +143892.181,E4 +0.000} C_DIS
LIN {X -189.772,Y +1119.341,Z +0.000,A -0.752,E1 -45.902,E3 +143905.719,E4 +0.000} C_DIS
LIN {X -189.097,Y +1124.276,Z +0.000,A -2.508,E1 -45.397,E3 +143912.451,E4 +0.000} C_DIS
LIN {X -187.410,Y +1129.069,Z +0.000,A -5.304,E1 -44.585,E3 +143919.624,E4 +0.000} C_DIS
LIN {X -183.899,Y +1134.873,Z +0.000,A -10.372,E1 -42.805,E3 +143929.630,E4 +0.000} C_DIS
LIN {X -179.711,Y +1140.065,Z +0.000,A -15.940,E1 -40.393,E3 +143940.416,E4 +0.000} C_DIS
LIN {X -176.763,Y +1143.197,Z +0.000,A -18.748,E1 -38.674,E3 +143948.154,E4 +0.000} C_DIS
LIN {X -172.185,Y +1147.423,Z +0.000,A -19.971,E1 -36.175,E3 +143960.884,E4 +0.000} C_DIS
LIN {X -165.999,Y +1152.127,Z +0.000,A -20.000,E1 -32.027,E3 +143980.642,E4 +0.000} C_DIS
LIN {X -160.138,Y +1155.667,Z +0.000,A -20.000,E1 -26.368,E3 +144005.012,E4 +0.000} C_DIS
LIN {X -155.625,Y +1157.756,Z +0.000,A -20.000,E1 -19.505,E3 +144033.688,E4 +0.000} C_DIS
LIN {X -153.552,Y +1158.113,Z +0.000,A -20.000,E1 -11.113,E3 +144069.439,E4 +0.000} C_DIS
LIN {X -156.311,Y +1155.540,Z +0.000,A -20.000,E1 -0.839,E3 +144112.799,E4 +0.000} C_DIS
LIN {X -161.281,Y +1151.851,Z +0.000,A -20.000,E1 +7.737,E3 +144142.698,E4 +0.000} C_DIS
LIN {X -167.493,Y +1147.157,Z +0.000,A -20.000,E1 +16.195,E3 +144167.137,E4 +0.000} C_DIS
LIN {X -173.235,Y +1142.221,Z +0.000,A -20.000,E1 +22.930,E3 +144184.439,E4 +0.000} C_DIS
LIN {X -181.123,Y +1133.734,Z +0.000,A -20.000,E1 +30.868,E3 +144205.195,E4 +0.000} C_DIS
LIN {X -189.654,Y +1120.856,Z +0.000,A -20.000,E1 +39.018,E3 +144227.209,E4 +0.000} C_DIS
LIN {X -195.246,Y +1107.046,Z +0.000,A -20.000,E1 +44.515,E3 +144245.111,E4 +0.000} C_DIS
LIN {X -198.051,Y +1092.368,Z +0.000,A -20.000,E1 +47.947,E3 +144261.637,E4 +0.000} C_DIS
LIN {X -198.143,Y +1081.370,Z +0.000,A -19.806,E1 +49.153,E3 +144273.498,E4 +0.000} C_DIS
LIN {X -197.177,Y +1073.569,Z +0.000,A -17.356,E1 +49.162,E3 +144282.082,E4 +0.000} C_DIS
LIN {X -195.448,Y +1066.139,Z +0.000,A -12.154,E1 +48.512,E3 +144290.677,E4 +0.000} C_DIS
LIN {X -193.346,Y +1058.941,Z +0.000,A -7.133,E1 +47.724,E3 +144299.557,E4 +0.000} C_DIS
LIN {X -191.781,Y +1050.839,Z +0.000,A -3.715,E1 +47.274,E3 +144309.890,E4 +0.000} C_DIS
LIN {X -190.795,Y +1039.355,Z +0.000,A -0.983,E1 +46.842,E3 +144324.550,E4 +0.000} C_DIS
LIN {X -190.395,Y +1028.856,Z +0.000,A -0.089,E1 +46.598,E3 +144337.944,E4 +0.000} C_DIS
LIN {X -190.239,Y +1018.851,Z +0.000,A -0.004,E1 +46.529,E3 +144350.712,E4 +0.000} C_DIS
LIN {X -190.161,Y +1004.975,Z +0.000,A +0.000,E1 +46.506,E3 +144368.426,E4 +0.000} C_DIS
LIN {X -190.142,Y +412.853,Z +0.000,A +0.000,E1 +46.501,E3 +145124.632,E4 +0.000} C_DIS
LIN {X -190.147,Y +401.077,Z +0.000,A +0.000,E1 +46.499,E3 +145139.673,E4 +0.000} C_DIS
LIN {X -190.159,Y +390.929,Z +0.000,A +0.000,E1 +46.494,E3 +145152.639,E4 +0.000} C_DIS
LIN {X -190.174,Y +383.973,Z +0.000,A +0.000,E1 +46.484,E3 +145161.532,E4 +0.000} C_DIS
LIN {X -190.200,Y +373.815,Z +0.000,A +0.000,E1 +46.448,E3 +145174.537,E4 +0.000} C_DIS
LIN {X -190.154,Y +361.003,Z +0.000,A +0.000,E1 +46.303,E3 +145191.031,E4 +0.000} C_DIS
LIN {X -189.772,Y +350.660,Z +0.000,A +0.049,E1 +45.996,E3 +145204.570,E4 +0.000} C_DIS
LIN {X -189.325,Y +346.917,Z +0.000,A +0.243,E1 +45.771,E3 +145209.639,E4 +0.000} C_DIS
LIN {X -188.196,Y +342.754,Z +0.000,A +1.966,E1 +45.249,E3 +145215.647,E4 +0.000} C_DIS
LIN {X -185.199,Y +337.023,Z +0.000,A +6.630,E1 +43.793,E3 +145225.021,E4 +0.000} C_DIS
LIN {X -181.141,Y +331.596,Z +0.000,A +12.274,E1 +41.569,E3 +145235.581,E4 +0.000} C_DIS
LIN {X -176.762,Y +326.804,Z +0.000,A +17.560,E1 +38.898,E3 +145247.005,E4 +0.000} C_DIS
LIN {X -172.184,Y +322.578,Z +0.000,A +19.859,E1 +36.197,E3 +145259.735,E4 +0.000} C_DIS
LIN {X -165.998,Y +317.874,Z +0.000,A +20.000,E1 +32.027,E3 +145279.493,E4 +0.000} C_DIS
LIN {X -160.137,Y +314.334,Z +0.000,A +20.000,E1 +26.368,E3 +145303.862,E4 +0.000} C_DIS
LIN {X -155.624,Y +312.245,Z +0.000,A +20.000,E1 +19.506,E3 +145332.538,E4 +0.000} C_DIS
LIN {X -153.557,Y +311.879,Z +0.000,A +20.000,E1 +11.113,E3 +145368.293,E4 +0.000} C_DIS
LIN {X -155.320,Y +313.348,Z +0.000,A +20.000,E1 +3.401,E3 +145401.477,E4 +0.000} C_DIS
LIN {X -160.005,Y +315.804,Z +0.000,A +20.000,E1 -4.720,E3 +145431.855,E4 +0.000} C_DIS
LIN {X -164.504,Y +318.255,Z +0.000,A +20.000,E1 -10.663,E3 +145451.224,E4 +0.000} C_DIS
LIN {X -170.340,Y +322.684,Z +0.000,A +20.000,E1 -17.457,E3 +145471.256,E4 +0.000} C_DIS
LIN {X -175.568,Y +329.106,Z +0.000,A +20.000,E1 -24.747,E3 +145488.490,E4 +0.000} C_DIS
LIN {X -184.074,Y +340.065,Z +0.000,A +20.000,E1 -33.664,E3 +145511.430,E4 +0.000} C_DIS
LIN {X -190.779,Y +351.388,Z +0.000,A +20.000,E1 -40.083,E3 +145529.208,E4 +0.000} C_DIS
LIN {X -195.254,Y +362.955,Z +0.000,A +20.000,E1 -44.515,E3 +145543.961,E4 +0.000} C_DIS
LIN {X -197.754,Y +374.780,Z +0.000,A +20.000,E1 -47.450,E3 +145557.383,E4 +0.000} C_DIS
LIN {X -198.310,Y +383.215,Z +0.000,A +19.956,E1 -48.698,E3 +145566.507,E4 +0.000} C_DIS
LIN {X -197.912,Y +391.275,Z +0.000,A +18.601,E1 -49.158,E3 +145575.225,E4 +0.000} C_DIS
LIN {X -196.679,Y +398.944,Z +0.000,A +13.989,E1 -48.784,E3 +145583.779,E4 +0.000} C_DIS
LIN {X -194.742,Y +406.288,Z +0.000,A +8.476,E1 -48.001,E3 +145592.462,E4 +0.000} C_DIS
LIN {X -192.748,Y +413.472,Z +0.000,A +3.905,E1 -47.267,E3 +145601.472,E4 +0.000} C_DIS
LIN {X -191.781,Y +419.162,Z +0.000,A +1.739,E1 -46.975,E3 +145608.740,E4 +0.000} C_DIS
LIN {X -190.795,Y +430.646,Z +0.000,A +0.152,E1 -46.707,E3 +145623.401,E4 +0.000} C_DIS
LIN {X -190.395,Y +441.145,Z +0.000,A +0.001,E1 -46.583,E3 +145636.794,E4 +0.000} C_DIS
LIN {X -190.239,Y +451.150,Z +0.000,A -0.000,E1 -46.528,E3 +145649.562,E4 +0.000} C_DIS
LIN {X -190.161,Y +465.026,Z +0.000,A -0.000,E1 -46.506,E3 +145667.277,E4 +0.000} C_DIS
LIN {X -190.142,Y +1057.148,Z +0.000,A -0.000,E1 -46.500,E3 +146423.483,E4 +0.000} C_DIS
LIN {X -190.147,Y +1068.924,Z +0.000,A -0.000,E1 -46.499,E3 +146438.524,E4 +0.000} C_DIS
LIN {X -190.159,Y +1079.072,Z +0.000,A -0.000,E1 -46.493,E3 +146451.489,E4 +0.000} C_DIS
LIN {X -190.174,Y +1086.028,Z +0.000,A -0.000,E1 -46.483,E3 +146460.383,E4 +0.000} C_DIS
LIN {X -190.200,Y +1096.186,Z +0.000,A -0.000,E1 -46.448,E3 +146473.387,E4 +0.000} C_DIS
LIN {X -190.154,Y +1108.998,Z +0.000,A -0.054,E1 -46.295,E3 +146489.882,E4 +0.000} C_DIS
LIN {X -189.772,Y +1119.341,Z +0.000,A -0.752,E1 -45.902,E3 +146503.420,E4 +0.000} C_DIS
LIN {X -189.097,Y +1124.276,Z +0.000,A -2.508,E1 -45.397,E3 +146510.152,E4 +0.000} C_DIS
LIN {X -187.410,Y +1129.069,Z +0.000,A -5.304,E1 -44.585,E3 +146517.325,E4 +0.000} C_DIS
LIN {X -183.899,Y +1134.873,Z +0.000,A -10.372,E1 -42.805,E3 +146527.331,E4 +0.000} C_DIS
LIN {X -179.711,Y +1140.065,Z +0.000,A -15.940,E1 -40.393,E3 +146538.117,E4 +0.000} C_DIS
LIN {X -176.763,Y +1143.197,Z +0.000,A -18.748,E1 -38.674,E3 +146545.855,E4 +0.000} C_DIS
LIN {X -172.185,Y +1147.423,Z +0.000,A -19.971,E1 -36.175,E3 +146558.585,E4 +0.000} C_DIS
LIN {X -165.999,Y +1152.127,Z +0.000,A -20.000,E1 -32.027,E3 +146578.343,E4 +0.000} C_DIS
LIN {X -160.138,Y +1155.667,Z +0.000,A -20.000,E1 -26.368,E3 +146602.713,E4 +0.000} C_DIS
LIN {X -155.625,Y +1157.756,Z +0.000,A -20.000,E1 -19.505,E3 +146631.389,E4 +0.000} C_DIS
LIN {X -153.552,Y +1158.113,Z +0.000,A -20.000,E1 -11.113,E3 +146667.140,E4 +0.000} C_DIS
LIN {X -156.311,Y +1155.540,Z +0.000,A -20.000,E1 -0.839,E3 +146710.500,E4 +0.000} C_DIS
LIN {X -161.281,Y +1151.851,Z +0.000,A -20.000,E1 +7.737,E3 +146740.399,E4 +0.000} C_DIS
LIN {X -167.493,Y +1147.157,Z +0.000,A -20.000,E1 +16.195,E3 +146764.838,E4 +0.000} C_DIS
LIN {X -173.235,Y +1142.221,Z +0.000,A -20.000,E1 +22.930,E3 +146782.140,E4 +0.000} C_DIS
LIN {X -181.123,Y +1133.734,Z +0.000,A -20.000,E1 +30.868,E3 +146802.896,E4 +0.000} C_DIS
LIN {X -189.654,Y +1120.856,Z +0.000,A -20.000,E1 +39.018,E3 +146824.910,E4 +0.000} C_DIS
LIN {X -195.246,Y +1107.046,Z +0.000,A -20.000,E1 +44.515,E3 +146842.812,E4 +0.000} C_DIS
LIN {X -198.051,Y +1092.368,Z +0.000,A -20.000,E1 +47.947,E3 +146859.338,E4 +0.000} C_DIS
LIN {X -198.143,Y +1081.370,Z +0.000,A -19.806,E1 +49.153,E3 +146871.199,E4 +0.000} C_DIS
LIN {X -197.177,Y +1073.569,Z +0.000,A -17.356,E1 +49.162,E3 +146879.783,E4 +0.000} C_DIS
LIN {X -195.448,Y +1066.139,Z +0.000,A -12.154,E1 +48.512,E3 +146888.378,E4 +0.000} C_DIS
LIN {X -193.346,Y +1058.941,Z +0.000,A -7.133,E1 +47.724,E3 +146897.258,E4 +0.000} C_DIS
LIN {X -191.781,Y +1050.839,Z +0.000,A -3.715,E1 +47.274,E3 +146907.591,E4 +0.000} C_DIS
LIN {X -190.795,Y +1039.355,Z +0.000,A -0.983,E1 +46.842,E3 +146922.251,E4 +0.000} C_DIS
LIN {X -190.395,Y +1028.856,Z +0.000,A -0.089,E1 +46.598,E3 +146935.645,E4 +0.000} C_DIS
LIN {X -190.239,Y +1018.851,Z +0.000,A -0.004,E1 +46.529,E3 +146948.413,E4 +0.000} C_DIS
LIN {X -190.161,Y +1004.975,Z +0.000,A +0.000,E1 +46.506,E3 +146966.127,E4 +0.000} C_DIS
LIN {X -190.142,Y +412.853,Z +0.000,A +0.000,E1 +46.501,E3 +147722.333,E4 +0.000} C_DIS
LIN {X -190.147,Y +401.077,Z +0.000,A +0.000,E1 +46.499,E3 +147737.374,E4 +0.000} C_DIS
LIN {X -190.159,Y +390.929,Z +0.000,A +0.000,E1 +46.494,E3 +147750.340,E4 +0.000} C_DIS
LIN {X -190.174,Y +383.973,Z +0.000,A +0.000,E1 +46.484,E3 +147759.233,E4 +0.000} C_DIS
LIN {X -190.200,Y +373.815,Z +0.000,A +0.000,E1 +46.448,E3 +147772.238,E4 +0.000} C_DIS
LIN {X -190.154,Y +361.003,Z +0.000,A +0.000,E1 +46.303,E3 +147788.732,E4 +0.000} C_DIS
LIN {X -189.772,Y +350.660,Z +0.000,A +0.049,E1 +45.996,E3 +147802.271,E4 +0.000} C_DIS
LIN {X -189.325,Y +346.917,Z +0.000,A +0.243,E1 +45.771,E3 +147807.340,E4 +0.000} C_DIS
LIN {X -188.196,Y +342.754,Z +0.000,A +1.966,E1 +45.249,E3 +147813.348,E4 +0.000} C_DIS
LIN {X -185.199,Y +337.023,Z +0.000,A +6.630,E1 +43.793,E3 +147822.722,E4 +0.000} C_DIS
LIN {X -181.141,Y +331.596,Z +0.000,A +12.274,E1 +41.569,E3 +147833.282,E4 +0.000} C_DIS
LIN {X -176.762,Y +326.804,Z +0.000,A +17.560,E1 +38.898,E3 +147844.706,E4 +0.000} C_DIS
LIN {X -172.184,Y +322.578,Z +0.000,A +19.859,E1 +36.197,E3 +147857.436,E4 +0.000} C_DIS
LIN {X -165.998,Y +317.874,Z +0.000,A +20.000,E1 +32.027,E3 +147877.194,E4 +0.000} C_DIS
LIN {X -160.137,Y +314.334,Z +0.000,A +20.000,E1 +26.368,E3 +147901.563,E4 +0.000} C_DIS
LIN {X -155.624,Y +312.245,Z +0.000,A +20.000,E1 +19.506,E3 +147930.239,E4 +0.000} C_DIS
LIN {X -153.557,Y +311.879,Z +0.000,A +20.000,E1 +11.113,E3 +147965.994,E4 +0.000} C_DIS
LIN {X -155.320,Y +313.348,Z +0.000,A +20.000,E1 +3.401,E3 +147999.178,E4 +0.000} C_DIS
LIN {X -160.005,Y +315.804,Z +0.000,A +20.000,E1 -4.720,E3 +148029.556,E4 +0.000} C_DIS
LIN {X -164.504,Y +318.255,Z +0.000,A +20.000,E1 -10.663,E3 +148048.925,E4 +0.000} C_DIS
LIN {X -170.340,Y +322.684,Z +0.000,A +20.000,E1 -17.457,E3 +148068.957,E4 +0.000} C_DIS
LIN {X -175.568,Y +329.106,Z +0.000,A +20.000,E1 -24.747,E3 +148086.191,E4 +0.000} C_DIS
LIN {X -184.074,Y +340.065,Z +0.000,A +20.000,E1 -33.664,E3 +148109.131,E4 +0.000} C_DIS
LIN {X -190.779,Y +351.388,Z +0.000,A +20.000,E1 -40.083,E3 +148126.909,E4 +0.000} C_DIS
LIN {X -195.254,Y +362.955,Z +0.000,A +20.000,E1 -44.515,E3 +148141.662,E4 +0.000} C_DIS
LIN {X -197.754,Y +374.780,Z +0.000,A +20.000,E1 -47.450,E3 +148155.084,E4 +0.000} C_DIS
LIN {X -198.310,Y +383.215,Z +0.000,A +19.956,E1 -48.698,E3 +148164.208,E4 +0.000} C_DIS
LIN {X -197.912,Y +391.275,Z +0.000,A +18.601,E1 -49.158,E3 +148172.926,E4 +0.000} C_DIS
LIN {X -196.679,Y +398.944,Z +0.000,A +13.989,E1 -48.784,E3 +148181.480,E4 +0.000} C_DIS
LIN {X -194.742,Y +406.288,Z +0.000,A +8.476,E1 -48.001,E3 +148190.163,E4 +0.000} C_DIS
LIN {X -192.748,Y +413.472,Z +0.000,A +3.905,E1 -47.267,E3 +148199.173,E4 +0.000} C_DIS
LIN {X -191.781,Y +419.162,Z +0.000,A +1.739,E1 -46.975,E3 +148206.441,E4 +0.000} C_DIS
LIN {X -190.795,Y +430.646,Z +0.000,A +0.152,E1 -46.707,E3 +148221.102,E4 +0.000} C_DIS
LIN {X -190.395,Y +441.145,Z +0.000,A +0.001,E1 -46.583,E3 +148234.495,E4 +0.000} C_DIS
LIN {X -190.239,Y +451.150,Z +0.000,A -0.000,E1 -46.528,E3 +148247.263,E4 +0.000} C_DIS
LIN {X -190.161,Y +465.026,Z +0.000,A -0.000,E1 -46.506,E3 +148264.978,E4 +0.000} C_DIS
LIN {X -190.142,Y +1057.148,Z +0.000,A -0.000,E1 -46.500,E3 +149021.184,E4 +0.000} C_DIS
LIN {X -190.147,Y +1068.924,Z +0.000,A -0.000,E1 -46.499,E3 +149036.225,E4 +0.000} C_DIS
LIN {X -190.159,Y +1079.072,Z +0.000,A -0.000,E1 -46.493,E3 +149049.190,E4 +0.000} C_DIS
LIN {X -190.174,Y +1086.028,Z +0.000,A -0.000,E1 -46.483,E3 +149058.084,E4 +0.000} C_DIS
LIN {X -190.200,Y +1096.186,Z +0.000,A -0.000,E1 -46.448,E3 +149071.088,E4 +0.000} C_DIS
LIN {X -190.154,Y +1108.998,Z +0.000,A -0.054,E1 -46.295,E3 +149087.583,E4 +0.000} C_DIS
LIN {X -189.772,Y +1119.341,Z +0.000,A -0.752,E1 -45.902,E3 +149101.121,E4 +0.000} C_DIS
LIN {X -189.097,Y +1124.276,Z +0.000,A -2.508,E1 -45.397,E3 +149107.853,E4 +0.000} C_DIS
LIN {X -187.410,Y +1129.069,Z +0.000,A -5.304,E1 -44.585,E3 +149115.026,E4 +0.000} C_DIS
LIN {X -183.899,Y +1134.873,Z +0.000,A -10.372,E1 -42.805,E3 +149125.032,E4 +0.000} C_DIS
LIN {X -179.711,Y +1140.065,Z +0.000,A -15.940,E1 -40.393,E3 +149135.818,E4 +0.000} C_DIS
LIN {X -176.763,Y +1143.197,Z +0.000,A -18.748,E1 -38.674,E3 +149143.556,E4 +0.000} C_DIS
LIN {X -172.185,Y +1147.423,Z +0.000,A -19.971,E1 -36.175,E3 +149156.286,E4 +0.000} C_DIS
LIN {X -165.999,Y +1152.127,Z +0.000,A -20.000,E1 -32.027,E3 +149176.044,E4 +0.000} C_DIS
LIN {X -160.138,Y +1155.667,Z +0.000,A -20.000,E1 -26.368,E3 +149200.414,E4 +0.000} C_DIS
LIN {X -155.625,Y +1157.756,Z +0.000,A -20.000,E1 -19.505,E3 +149229.090,E4 +0.000} C_DIS
LIN {X -153.552,Y +1158.113,Z +0.000,A -20.000,E1 -11.113,E3 +149264.841,E4 +0.000} C_DIS
LIN {X -156.311,Y +1155.540,Z +0.000,A -20.000,E1 -0.839,E3 +149308.201,E4 +0.000} C_DIS
LIN {X -161.281,Y +1151.851,Z +0.000,A -20.000,E1 +7.737,E3 +149338.100,E4 +0.000} C_DIS
LIN {X -167.493,Y +1147.157,Z +0.000,A -20.000,E1 +16.195,E3 +149362.539,E4 +0.000} C_DIS
LIN {X -173.235,Y +1142.221,Z +0.000,A -20.000,E1 +22.930,E3 +149379.841,E4 +0.000} C_DIS
LIN {X -181.123,Y +1133.734,Z +0.000,A -20.000,E1 +30.868,E3 +149400.597,E4 +0.000} C_DIS
LIN {X -189.654,Y +1120.856,Z +0.000,A -20.000,E1 +39.018,E3 +149422.611,E4 +0.000} C_DIS
LIN {X -195.246,Y +1107.046,Z +0.000,A -20.000,E1 +44.515,E3 +149440.513,E4 +0.000} C_DIS
LIN {X -198.051,Y +1092.368,Z +0.000,A -20.000,E1 +47.947,E3 +149457.039,E4 +0.000} C_DIS
LIN {X -198.143,Y +1081.370,Z +0.000,A -19.806,E1 +49.153,E3 +149468.900,E4 +0.000} C_DIS
LIN {X -197.177,Y +1073.569,Z +0.000,A -17.356,E1 +49.162,E3 +149477.484,E4 +0.000} C_DIS
LIN {X -195.448,Y +1066.139,Z +0.000,A -12.154,E1 +48.512,E3 +149486.079,E4 +0.000} C_DIS
LIN {X -193.346,Y +1058.941,Z +0.000,A -7.133,E1 +47.724,E3 +149494.959,E4 +0.000} C_DIS
LIN {X -191.781,Y +1050.839,Z +0.000,A -3.715,E1 +47.274,E3 +149505.292,E4 +0.000} C_DIS
LIN {X -190.795,Y +1039.355,Z +0.000,A -0.983,E1 +46.842,E3 +149519.952,E4 +0.000} C_DIS
LIN {X -190.395,Y +1028.856,Z +0.000,A -0.089,E1 +46.598,E3 +149533.346,E4 +0.000} C_DIS
LIN {X -190.239,Y +1018.851,Z +0.000,A -0.004,E1 +46.529,E3 +149546.114,E4 +0.000} C_DIS
LIN {X -190.161,Y +1004.975,Z +0.000,A +0.000,E1 +46.506,E3 +149563.828,E4 +0.000} C_DIS
LIN {X -190.142,Y +412.853,Z +0.000,A +0.000,E1 +46.501,E3 +150320.034,E4 +0.000} C_DIS
LIN {X -190.147,Y +401.077,Z +0.000,A +0.000,E1 +46.499,E3 +150335.075,E4 +0.000} C_DIS
LIN {X -190.159,Y +390.929,Z +0.000,A +0.000,E1 +46.494,E3 +150348.041,E4 +0.000} C_DIS
LIN {X -190.174,Y +383.973,Z +0.000,A +0.000,E1 +46.484,E3 +150356.934,E4 +0.000} C_DIS
LIN {X -190.200,Y +373.815,Z +0.000,A +0.000,E1 +46.448,E3 +150369.939,E4 +0.000} C_DIS
LIN {X -190.154,Y +361.003,Z +0.000,A +0.000,E1 +46.303,E3 +150386.433,E4 +0.000} C_DIS
LIN {X -189.772,Y +350.660,Z +0.000,A +0.049,E1 +45.996,E3 +150399.972,E4 +0.000} C_DIS
LIN {X -189.325,Y +346.917,Z +0.000,A +0.243,E1 +45.771,E3 +150405.041,E4 +0.000} C_DIS
LIN {X -188.196,Y +342.754,Z +0.000,A +1.966,E1 +45.249,E3 +150411.049,E4 +0.000} C_DIS
LIN {X -185.199,Y +337.023,Z +0.000,A +6.630,E1 +43.793,E3 +150420.423,E4 +0.000} C_DIS
LIN {X -181.141,Y +331.596,Z +0.000,A +12.274,E1 +41.569,E3 +150430.983,E4 +0.000} C_DIS
LIN {X -176.762,Y +326.804,Z +0.000,A +17.560,E1 +38.898,E3 +150442.407,E4 +0.000} C_DIS
LIN {X -172.184,Y +322.578,Z +0.000,A +19.859,E1 +36.197,E3 +150455.137,E4 +0.000} C_DIS
LIN {X -165.998,Y +317.874,Z +0.000,A +20.000,E1 +32.027,E3 +150474.895,E4 +0.000} C_DIS
LIN {X -160.137,Y +314.334,Z +0.000,A +20.000,E1 +26.368,E3 +150499.264,E4 +0.000} C_DIS
LIN {X -155.624,Y +312.245,Z +0.000,A +20.000,E1 +19.506,E3 +150527.940,E4 +0.000} C_DIS
LIN {X -153.557,Y +311.879,Z +0.000,A +20.000,E1 +11.113,E3 +150563.695,E4 +0.000} C_DIS
LIN {X -155.320,Y +313.348,Z +0.000,A +20.000,E1 +3.401,E3 +150596.879,E4 +0.000} C_DIS
LIN {X -160.005,Y +315.804,Z +0.000,A +20.000,E1 -4.720,E3 +150627.257,E4 +0.000} C_DIS
LIN {X -164.504,Y +318.255,Z +0.000,A +20.000,E1 -10.663,E3 +150646.626,E4 +0.000} C_DIS
LIN {X -170.340,Y +322.684,Z +0.000,A +20.000,E1 -17.457,E3 +150666.658,E4 +0.000} C_DIS
LIN {X -175.568,Y +329.106,Z +0.000,A +20.000,E1 -24.747,E3 +150683.892,E4 +0.000} C_DIS
LIN {X -184.074,Y +340.065,Z +0.000,A +20.000,E1 -33.664,E3 +150706.832,E4 +0.000} C_DIS
LIN {X -190.779,Y +351.388,Z +0.000,A +20.000,E1 -40.083,E3 +150724.610,E4 +0.000} C_DIS
LIN {X -195.254,Y +362.955,Z +0.000,A +20.000,E1 -44.515,E3 +150739.363,E4 +0.000} C_DIS
LIN {X -197.754,Y +374.780,Z +0.000,A +20.000,E1 -47.450,E3 +150752.785,E4 +0.000} C_DIS
LIN {X -198.310,Y +383.215,Z +0.000,A +19.956,E1 -48.698,E3 +150761.909,E4 +0.000} C_DIS
LIN {X -197.912,Y +391.275,Z +0.000,A +18.601,E1 -49.158,E3 +150770.627,E4 +0.000} C_DIS
LIN {X -196.679,Y +398.944,Z +0.000,A +13.989,E1 -48.784,E3 +150779.181,E4 +0.000} C_DIS
LIN {X -194.742,Y +406.288,Z +0.000,A +8.476,E1 -48.001,E3 +150787.864,E4 +0.000} C_DIS
LIN {X -192.748,Y +413.472,Z +0.000,A +3.905,E1 -47.267,E3 +150796.874,E4 +0.000} C_DIS
LIN {X -191.781,Y +419.162,Z +0.000,A +1.739,E1 -46.975,E3 +150804.142,E4 +0.000} C_DIS
LIN {X -190.795,Y +430.646,Z +0.000,A +0.152,E1 -46.707,E3 +150818.803,E4 +0.000} C_DIS
LIN {X -190.395,Y +441.145,Z +0.000,A +0.001,E1 -46.583,E3 +150832.196,E4 +0.000} C_DIS
LIN {X -190.239,Y +451.150,Z +0.000,A -0.000,E1 -46.528,E3 +150844.964,E4 +0.000} C_DIS
LIN {X -190.161,Y +465.026,Z +0.000,A -0.000,E1 -46.506,E3 +150862.679,E4 +0.000} C_DIS
LIN {X -190.142,Y +1057.148,Z +0.000,A -0.000,E1 -46.500,E3 +151618.885,E4 +0.000} C_DIS
LIN {X -190.147,Y +1068.924,Z +0.000,A -0.000,E1 -46.499,E3 +151633.926,E4 +0.000} C_DIS
LIN {X -190.159,Y +1079.072,Z +0.000,A -0.000,E1 -46.493,E3 +151646.891,E4 +0.000} C_DIS
LIN {X -190.174,Y +1086.028,Z +0.000,A -0.000,E1 -46.483,E3 +151655.785,E4 +0.000} C_DIS
LIN {X -190.200,Y +1096.186,Z +0.000,A -0.000,E1 -46.448,E3 +151668.789,E4 +0.000} C_DIS
LIN {X -190.154,Y +1108.998,Z +0.000,A -0.054,E1 -46.295,E3 +151685.284,E4 +0.000} C_DIS
LIN {X -189.772,Y +1119.341,Z +0.000,A -0.752,E1 -45.902,E3 +151698.822,E4 +0.000} C_DIS
LIN {X -189.097,Y +1124.276,Z +0.000,A -2.508,E1 -45.397,E3 +151705.554,E4 +0.000} C_DIS
LIN {X -187.410,Y +1129.069,Z +0.000,A -5.304,E1 -44.585,E3 +151712.727,E4 +0.000} C_DIS
LIN {X -183.899,Y +1134.873,Z +0.000,A -10.372,E1 -42.805,E3 +151722.733,E4 +0.000} C_DIS
LIN {X -179.711,Y +1140.065,Z +0.000,A -15.940,E1 -40.393,E3 +151733.519,E4 +0.000} C_DIS
LIN {X -176.763,Y +1143.197,Z +0.000,A -18.748,E1 -38.674,E3 +151741.257,E4 +0.000} C_DIS
LIN {X -172.185,Y +1147.423,Z +0.000,A -19.971,E1 -36.175,E3 +151753.987,E4 +0.000} C_DIS
LIN {X -165.999,Y +1152.127,Z +0.000,A -20.000,E1 -32.027,E3 +151773.745,E4 +0.000} C_DIS
LIN {X -160.138,Y +1155.667,Z +0.000,A -20.000,E1 -26.368,E3 +151798.115,E4 +0.000} C_DIS
LIN {X -155.625,Y +1157.756,Z +0.000,A -20.000,E1 -19.505,E3 +151826.791,E4 +0.000} C_DIS
LIN {X -153.552,Y +1158.113,Z +0.000,A -20.000,E1 -11.113,E3 +151862.542,E4 +0.000} C_DIS
LIN {X -156.311,Y +1155.540,Z +0.000,A -20.000,E1 -0.839,E3 +151905.902,E4 +0.000} C_DIS
LIN {X -161.281,Y +1151.851,Z +0.000,A -20.000,E1 +7.737,E3 +151935.801,E4 +0.000} C_DIS
LIN {X -167.493,Y +1147.157,Z +0.000,A -20.000,E1 +16.195,E3 +151960.240,E4 +0.000} C_DIS
LIN {X -173.235,Y +1142.221,Z +0.000,A -20.000,E1 +22.930,E3 +151977.542,E4 +0.000} C_DIS
LIN {X -181.123,Y +1133.734,Z +0.000,A -20.000,E1 +30.868,E3 +151998.298,E4 +0.000} C_DIS
LIN {X -189.654,Y +1120.856,Z +0.000,A -20.000,E1 +39.018,E3 +152020.312,E4 +0.000} C_DIS
LIN {X -195.246,Y +1107.046,Z +0.000,A -20.000,E1 +44.515,E3 +152038.214,E4 +0.000} C_DIS
LIN {X -198.051,Y +1092.368,Z +0.000,A -20.000,E1 +47.947,E3 +152054.740,E4 +0.000} C_DIS
LIN {X -198.143,Y +1081.370,Z +0.000,A -19.806,E1 +49.153,E3 +152066.601,E4 +0.000} C_DIS
LIN {X -197.177,Y +1073.569,Z +0.000,A -17.356,E1 +49.162,E3 +152075.185,E4 +0.000} C_DIS
LIN {X -195.448,Y +1066.139,Z +0.000,A -12.154,E1 +48.512,E3 +152083.780,E4 +0.000} C_DIS
LIN {X -193.346,Y +1058.941,Z +0.000,A -7.133,E1 +47.724,E3 +152092.660,E4 +0.000} C_DIS
LIN {X -191.781,Y +1050.839,Z +0.000,A -3.715,E1 +47.274,E3 +152102.993,E4 +0.000} C_DIS
LIN {X -190.795,Y +1039.355,Z +0.000,A -0.983,E1 +46.842,E3 +152117.653,E4 +0.000} C_DIS
LIN {X -190.395,Y +1028.856,Z +0.000,A -0.089,E1 +46.598,E3 +152131.047,E4 +0.000} C_DIS
LIN {X -190.239,Y +1018.851,Z +0.000,A -0.004,E1 +46.529,E3 +152143.815,E4 +0.000} C_DIS
LIN {X -190.161,Y +1004.975,Z +0.000,A +0.000,E1 +46.506,E3 +152161.529,E4 +0.000} C_DIS
LIN {X -190.142,Y +412.853,Z +0.000,A +0.000,E1 +46.501,E3 +152917.735,E4 +0.000} C_DIS
LIN {X -190.147,Y +401.077,Z +0.000,A +0.000,E1 +46.499,E3 +152932.776,E4 +0.000} C_DIS
LIN {X -190.159,Y +390.929,Z +0.000,A +0.000,E1 +46.494,E3 +152945.742,E4 +0.000} C_DIS
LIN {X -190.174,Y +383.973,Z +0.000,A +0.000,E1 +46.484,E3 +152954.635,E4 +0.000} C_DIS
LIN {X -190.200,Y +373.815,Z +0.000,A +0.000,E1 +46.448,E3 +152967.640,E4 +0.000} C_DIS
LIN {X -190.154,Y +361.003,Z +0.000,A +0.000,E1 +46.303,E3 +152984.134,E4 +0.000} C_DIS
LIN {X -189.772,Y +350.660,Z +0.000,A +0.049,E1 +45.996,E3 +152997.673,E4 +0.000} C_DIS
LIN {X -189.325,Y +346.917,Z +0.000,A +0.243,E1 +45.771,E3 +153002.742,E4 +0.000} C_DIS
LIN {X -188.196,Y +342.754,Z +0.000,A +1.966,E1 +45.249,E3 +153008.750,E4 +0.000} C_DIS
LIN {X -185.199,Y +337.023,Z +0.000,A +6.630,E1 +43.793,E3 +153018.124,E4 +0.000} C_DIS
LIN {X -181.141,Y +331.596,Z +0.000,A +12.274,E1 +41.569,E3 +153028.684,E4 +0.000} C_DIS
LIN {X -176.762,Y +326.804,Z +0.000,A +17.560,E1 +38.898,E3 +153040.108,E4 +0.000} C_DIS
LIN {X -172.184,Y +322.578,Z +0.000,A +19.859,E1 +36.197,E3 +153052.838,E4 +0.000} C_DIS
LIN {X -165.998,Y +317.874,Z +0.000,A +20.000,E1 +32.027,E3 +153072.596,E4 +0.000} C_DIS
LIN {X -160.137,Y +314.334,Z +0.000,A +20.000,E1 +26.368,E3 +153096.965,E4 +0.000} C_DIS
LIN {X -155.624,Y +312.245,Z +0.000,A +20.000,E1 +19.506,E3 +153125.641,E4 +0.000} C_DIS
LIN {X -153.557,Y +311.879,Z +0.000,A +20.000,E1 +11.113,E3 +153161.396,E4 +0.000} C_DIS
LIN {X -155.320,Y +313.348,Z +0.000,A +20.000,E1 +3.401,E3 +153194.580,E4 +0.000} C_DIS
LIN {X -160.005,Y +315.804,Z +0.000,A +20.000,E1 -4.720,E3 +153224.958,E4 +0.000} C_DIS
LIN {X -164.504,Y +318.255,Z +0.000,A +20.000,E1 -10.663,E3 +153244.327,E4 +0.000} C_DIS
LIN {X -170.340,Y +322.684,Z +0.000,A +20.000,E1 -17.457,E3 +153264.359,E4 +0.000} C_DIS
LIN {X -175.568,Y +329.106,Z +0.000,A +20.000,E1 -24.747,E3 +153281.593,E4 +0.000} C_DIS
LIN {X -184.074,Y +340.065,Z +0.000,A +20.000,E1 -33.664,E3 +153304.533,E4 +0.000} C_DIS
LIN {X -190.779,Y +351.388,Z +0.000,A +20.000,E1 -40.083,E3 +153322.311,E4 +0.000} C_DIS
LIN {X -195.254,Y +362.955,Z +0.000,A +20.000,E1 -44.515,E3 +153337.064,E4 +0.000} C_DIS
LIN {X -197.754,Y +374.780,Z +0.000,A +20.000,E1 -47.450,E3 +153350.486,E4 +0.000} C_DIS
LIN {X -198.310,Y +383.215,Z +0.000,A +19.956,E1 -48.698,E3 +153359.610,E4 +0.000} C_DIS
LIN {X -197.912,Y +391.275,Z +0.000,A +18.601,E1 -49.158,E3 +153368.328,E4 +0.000} C_DIS
LIN {X -196.679,Y +398.944,Z +0.000,A +13.989,E1 -48.784,E3 +153376.882,E4 +0.000} C_DIS
LIN {X -194.742,Y +406.288,Z +0.000,A +8.476,E1 -48.001,E3 +153385.565,E4 +0.000} C_DIS
LIN {X -192.748,Y +413.472,Z +0.000,A +3.905,E1 -47.267,E3 +153394.575,E4 +0.000} C_DIS
LIN {X -191.781,Y +419.162,Z +0.000,A +1.739,E1 -46.975,E3 +153401.843,E4 +0.000} C_DIS
LIN {X -190.795,Y +430.646,Z +0.000,A +0.152,E1 -46.707,E3 +153416.504,E4 +0.000} C_DIS
LIN {X -190.395,Y +441.145,Z +0.000,A +0.001,E1 -46.583,E3 +153429.897,E4 +0.000} C_DIS
LIN {X -190.239,Y +451.150,Z +0.000,A -0.000,E1 -46.528,E3 +153442.665,E4 +0.000} C_DIS
LIN {X -190.161,Y +465.026,Z +0.000,A -0.000,E1 -46.506,E3 +153460.380,E4 +0.000} C_DIS
LIN {X -190.142,Y +1057.148,Z +0.000,A -0.000,E1 -46.500,E3 +154216.586,E4 +0.000} C_DIS
LIN {X -190.147,Y +1068.924,Z +0.000,A -0.000,E1 -46.499,E3 +154231.627,E4 +0.000} C_DIS
LIN {X -190.159,Y +1079.072,Z +0.000,A -0.000,E1 -46.493,E3 +154244.592,E4 +0.000} C_DIS
LIN {X -190.174,Y +1086.028,Z +0.000,A -0.000,E1 -46.483,E3 +154253.486,E4 +0.000} C_DIS
LIN {X -190.200,Y +1096.186,Z +0.000,A -0.000,E1 -46.448,E3 +154266.490,E4 +0.000} C_DIS
LIN {X -190.154,Y +1108.998,Z +0.000,A -0.054,E1 -46.295,E3 +154282.985,E4 +0.000} C_DIS
LIN {X -189.772,Y +1119.341,Z +0.000,A -0.752,E1 -45.902,E3 +154296.523,E4 +0.000} C_DIS
LIN {X -189.097,Y +1124.276,Z +0.000,A -2.508,E1 -45.397,E3 +154303.255,E4 +0.000} C_DIS
LIN {X -187.410,Y +1129.069,Z +0.000,A -5.304,E1 -44.585,E3 +154310.428,E4 +0.000} C_DIS
LIN {X -183.899,Y +1134.873,Z +0.000,A -10.372,E1 -42.805,E3 +154320.434,E4 +0.000} C_DIS
LIN {X -179.711,Y +1140.065,Z +0.000,A -15.940,E1 -40.393,E3 +154331.220,E4 +0.000} C_DIS
LIN {X -176.763,Y +1143.197,Z +0.000,A -18.748,E1 -38.674,E3 +154338.958,E4 +0.000} C_DIS
LIN {X -172.185,Y +1147.423,Z +0.000,A -19.971,E1 -36.175,E3 +154351.688,E4 +0.000} C_DIS
LIN {X -165.999,Y +1152.127,Z +0.000,A -20.000,E1 -32.027,E3 +154371.446,E4 +0.000} C_DIS
LIN {X -160.138,Y +1155.667,Z +0.000,A -20.000,E1 -26.368,E3 +154395.816,E4 +0.000} C_DIS
LIN {X -155.625,Y +1157.756,Z +0.000,A -20.000,E1 -19.505,E3 +154424.492,E4 +0.000} C_DIS
LIN {X -153.552,Y +1158.113,Z +0.000,A -20.000,E1 -11.113,E3 +154460.243,E4 +0.000} C_DIS
LIN {X -156.311,Y +1155.540,Z +0.000,A -20.000,E1 -0.839,E3 +154503.603,E4 +0.000} C_DIS
LIN {X -161.281,Y +1151.851,Z +0.000,A -20.000,E1 +7.737,E3 +154533.502,E4 +0.000} C_DIS
LIN {X -167.493,Y +1147.157,Z +0.000,A -20.000,E1 +16.195,E3 +154557.941,E4 +0.000} C_DIS
LIN {X -173.235,Y +1142.221,Z +0.000,A -20.000,E1 +22.930,E3 +154575.243,E4 +0.000} C_DIS
LIN {X -181.123,Y +1133.734,Z +0.000,A -20.000,E1 +30.868,E3 +154595.999,E4 +0.000} C_DIS
LIN {X -189.654,Y +1120.856,Z +0.000,A -20.000,E1 +39.018,E3 +154618.013,E4 +0.000} C_DIS
LIN {X -195.246,Y +1107.046,Z +0.000,A -20.000,E1 +44.515,E3 +154635.915,E4 +0.000} C_DIS
LIN {X -198.051,Y +1092.368,Z +0.000,A -20.000,E1 +47.947,E3 +154652.441,E4 +0.000} C_DIS
LIN {X -198.143,Y +1081.370,Z +0.000,A -19.806,E1 +49.153,E3 +154664.302,E4 +0.000} C_DIS
LIN {X -197.177,Y +1073.569,Z +0.000,A -17.356,E1 +49.162,E3 +154672.886,E4 +0.000} C_DIS
LIN {X -195.448,Y +1066.139,Z +0.000,A -12.154,E1 +48.512,E3 +154681.481,E4 +0.000} C_DIS
LIN {X -193.346,Y +1058.941,Z +0.000,A -7.133,E1 +47.724,E3 +154690.361,E4 +0.000} C_DIS
LIN {X -191.781,Y +1050.839,Z +0.000,A -3.715,E1 +47.274,E3 +154700.694,E4 +0.000} C_DIS
LIN {X -190.795,Y +1039.355,Z +0.000,A -0.983,E1 +46.842,E3 +154715.354,E4 +0.000} C_DIS
LIN {X -190.395,Y +1028.856,Z +0.000,A -0.089,E1 +46.598,E3 +154728.748,E4 +0.000} C_DIS
LIN {X -190.239,Y +1018.851,Z +0.000,A -0.004,E1 +46.529,E3 +154741.516,E4 +0.000} C_DIS
LIN {X -190.161,Y +1004.975,Z +0.000,A +0.000,E1 +46.506,E3 +154759.230,E4 +0.000} C_DIS
LIN {X -190.142,Y +412.853,Z +0.000,A +0.000,E1 +46.501,E3 +155515.436,E4 +0.000} C_DIS
LIN {X -190.147,Y +401.077,Z +0.000,A +0.000,E1 +46.499,E3 +155530.477,E4 +0.000} C_DIS
LIN {X -190.159,Y +390.929,Z +0.000,A +0.000,E1 +46.494,E3 +155543.443,E4 +0.000} C_DIS
LIN {X -190.174,Y +383.973,Z +0.000,A +0.000,E1 +46.484,E3 +155552.336,E4 +0.000} C_DIS
LIN {X -190.200,Y +373.815,Z +0.000,A +0.000,E1 +46.448,E3 +155565.341,E4 +0.000} C_DIS
LIN {X -190.154,Y +361.003,Z +0.000,A +0.000,E1 +46.303,E3 +155581.835,E4 +0.000} C_DIS
LIN {X -189.772,Y +350.660,Z +0.000,A +0.049,E1 +45.996,E3 +155595.374,E4 +0.000} C_DIS
LIN {X -189.325,Y +346.917,Z +0.000,A +0.243,E1 +45.771,E3 +155600.443,E4 +0.000} C_DIS
LIN {X -188.196,Y +342.754,Z +0.000,A +1.966,E1 +45.249,E3 +155606.451,E4 +0.000} C_DIS
LIN {X -185.199,Y +337.023,Z +0.000,A +6.630,E1 +43.793,E3 +155615.825,E4 +0.000} C_DIS
LIN {X -181.141,Y +331.596,Z +0.000,A +12.274,E1 +41.569,E3 +155626.385,E4 +0.000} C_DIS
LIN {X -176.762,Y +326.804,Z +0.000,A +17.560,E1 +38.898,E3 +155637.809,E4 +0.000} C_DIS
LIN {X -172.184,Y +322.578,Z +0.000,A +19.859,E1 +36.197,E3 +155650.539,E4 +0.000} C_DIS
LIN {X -165.998,Y +317.874,Z +0.000,A +20.000,E1 +32.027,E3 +155670.297,E4 +0.000} C_DIS
LIN {X -160.137,Y +314.334,Z +0.000,A +20.000,E1 +26.368,E3 +155694.666,E4 +0.000} C_DIS
LIN {X -155.624,Y +312.245,Z +0.000,A +20.000,E1 +19.506,E3 +155723.342,E4 +0.000} C_DIS
LIN {X -153.557,Y +311.879,Z +0.000,A +20.000,E1 +11.113,E3 +155759.097,E4 +0.000} C_DIS
LIN {X -155.320,Y +313.348,Z +0.000,A +20.000,E1 +3.401,E3 +155792.281,E4 +0.000} C_DIS
LIN {X -160.005,Y +315.804,Z +0.000,A +20.000,E1 -4.720,E3 +155822.659,E4 +0.000} C_DIS
LIN {X -164.504,Y +318.255,Z +0.000,A +20.000,E1 -10.663,E3 +155842.028,E4 +0.000} C_DIS
LIN {X -170.340,Y +322.684,Z +0.000,A +20.000,E1 -17.457,E3 +155862.060,E4 +0.000} C_DIS
LIN {X -175.568,Y +329.106,Z +0.000,A +20.000,E1 -24.747,E3 +155879.294,E4 +0.000} C_DIS
LIN {X -184.074,Y +340.065,Z +0.000,A +20.000,E1 -33.664,E3 +155902.234,E4 +0.000} C_DIS
LIN {X -190.779,Y +351.388,Z +0.000,A +20.000,E1 -40.083,E3 +155920.012,E4 +0.000} C_DIS
LIN {X -195.254,Y +362.955,Z +0.000,A +20.000,E1 -44.515,E3 +155934.765,E4 +0.000} C_DIS
LIN {X -197.754,Y +374.780,Z +0.000,A +20.000,E1 -47.450,E3 +155948.187,E4 +0.000} C_DIS
LIN {X -198.310,Y +383.215,Z +0.000,A +19.956,E1 -48.698,E3 +155957.311,E4 +0.000} C_DIS
LIN {X -197.912,Y +391.275,Z +0.000,A +18.601,E1 -49.158,E3 +155966.029,E4 +0.000} C_DIS
LIN {X -196.679,Y +398.944,Z +0.000,A +13.989,E1 -48.784,E3 +155974.583,E4 +0.000} C_DIS
LIN {X -194.742,Y +406.288,Z +0.000,A +8.476,E1 -48.001,E3 +155983.266,E4 +0.000} C_DIS
LIN {X -192.748,Y +413.472,Z +0.000,A +3.905,E1 -47.267,E3 +155992.276,E4 +0.000} C_DIS
LIN {X -191.781,Y +419.162,Z +0.000,A +1.739,E1 -46.975,E3 +155999.544,E4 +0.000} C_DIS
LIN {X -190.795,Y +430.646,Z +0.000,A +0.152,E1 -46.707,E3 +156014.205,E4 +0.000} C_DIS
LIN {X -190.395,Y +441.145,Z +0.000,A +0.001,E1 -46.583,E3 +156027.598,E4 +0.000} C_DIS
LIN {X -190.239,Y +451.150,Z +0.000,A -0.000,E1 -46.528,E3 +156040.366,E4 +0.000} C_DIS
LIN {X -190.161,Y +465.026,Z +0.000,A -0.000,E1 -46.506,E3 +156058.081,E4 +0.000} C_DIS
LIN {X -190.142,Y +1057.148,Z +0.000,A -0.000,E1 -46.500,E3 +156814.287,E4 +0.000} C_DIS
LIN {X -190.147,Y +1068.924,Z +0.000,A -0.000,E1 -46.499,E3 +156829.328,E4 +0.000} C_DIS
LIN {X -190.159,Y +1079.072,Z +0.000,A -0.000,E1 -46.493,E3 +156842.293,E4 +0.000} C_DIS
LIN {X -190.174,Y +1086.028,Z +0.000,A -0.000,E1 -46.483,E3 +156851.187,E4 +0.000} C_DIS
LIN {X -190.200,Y +1096.186,Z +0.000,A -0.000,E1 -46.448,E3 +156864.191,E4 +0.000} C_DIS
LIN {X -190.154,Y +1108.998,Z +0.000,A -0.054,E1 -46.295,E3 +156880.686,E4 +0.000} C_DIS
LIN {X -189.772,Y +1119.341,Z +0.000,A -0.752,E1 -45.902,E3 +156894.224,E4 +0.000} C_DIS
LIN {X -189.097,Y +1124.276,Z +0.000,A -2.508,E1 -45.397,E3 +156900.956,E4 +0.000} C_DIS
LIN {X -187.410,Y +1129.069,Z +0.000,A -5.304,E1 -44.585,E3 +156908.129,E4 +0.000} C_DIS
LIN {X -183.899,Y +1134.873,Z +0.000,A -10.372,E1 -42.805,E3 +156918.135,E4 +0.000} C_DIS
LIN {X -179.711,Y +1140.065,Z +0.000,A -15.940,E1 -40.393,E3 +156928.921,E4 +0.000} C_DIS
LIN {X -176.763,Y +1143.197,Z +0.000,A -18.748,E1 -38.674,E3 +156936.659,E4 +0.000} C_DIS
LIN {X -172.185,Y +1147.423,Z +0.000,A -19.971,E1 -36.175,E3 +156949.389,E4 +0.000} C_DIS
LIN {X -165.999,Y +1152.127,Z +0.000,A -20.000,E1 -32.027,E3 +156969.147,E4 +0.000} C_DIS
LIN {X -160.138,Y +1155.667,Z +0.000,A -20.000,E1 -26.368,E3 +156993.517,E4 +0.000} C_DIS
LIN {X -155.625,Y +1157.756,Z +0.000,A -20.000,E1 -19.505,E3 +157022.193,E4 +0.000} C_DIS
LIN {X -153.552,Y +1158.113,Z +0.000,A -20.000,E1 -11.113,E3 +157057.944,E4 +0.000} C_DIS
LIN {X -156.311,Y +1155.540,Z +0.000,A -20.000,E1 -0.839,E3 +157101.304,E4 +0.000} C_DIS
LIN {X -161.281,Y +1151.851,Z +0.000,A -20.000,E1 +7.737,E3 +157131.203,E4 +0.000} C_DIS
LIN {X -167.493,Y +1147.157,Z +0.000,A -20.000,E1 +16.195,E3 +157155.642,E4 +0.000} C_DIS
LIN {X -173.235,Y +1142.221,Z +0.000,A -20.000,E1 +22.930,E3 +157172.944,E4 +0.000} C_DIS
LIN {X -181.123,Y +1133.734,Z +0.000,A -20.000,E1 +30.868,E3 +157193.700,E4 +0.000} C_DIS
LIN {X -189.654,Y +1120.856,Z +0.000,A -20.000,E1 +39.018,E3 +157215.714,E4 +0.000} C_DIS
LIN {X -195.246,Y +1107.046,Z +0.000,A -20.000,E1 +44.515,E3 +157233.616,E4 +0.000} C_DIS
LIN {X -198.051,Y +1092.368,Z +0.000,A -20.000,E1 +47.947,E3 +157250.142,E4 +0.000} C_DIS
LIN {X -198.143,Y +1081.370,Z +0.000,A -19.806,E1 +49.153,E3 +157262.003,E4 +0.000} C_DIS
LIN {X -197.177,Y +1073.569,Z +0.000,A -17.356,E1 +49.162,E3 +157270.587,E4 +0.000} C_DIS
LIN {X -195.448,Y +1066.139,Z +0.000,A -12.154,E1 +48.512,E3 +157279.182,E4 +0.000} C_DIS
LIN {X -193.346,Y +1058.941,Z +0.000,A -7.133,E1 +47.724,E3 +157288.062,E4 +0.000} C_DIS
LIN {X -191.781,Y +1050.839,Z +0.000,A -3.715,E1 +47.274,E3 +157298.395,E4 +0.000} C_DIS
LIN {X -190.795,Y +1039.355,Z +0.000,A -0.983,E1 +46.842,E3 +157313.055,E4 +0.000} C_DIS
LIN {X -190.395,Y +1028.856,Z +0.000,A -0.089,E1 +46.598,E3 +157326.449,E4 +0.000} C_DIS
LIN {X -190.239,Y +1018.851,Z +0.000,A -0.004,E1 +46.529,E3 +157339.217,E4 +0.000} C_DIS
LIN {X -190.161,Y +1004.975,Z +0.000,A +0.000,E1 +46.506,E3 +157356.931,E4 +0.000} C_DIS
LIN {X -190.142,Y +412.853,Z +0.000,A +0.000,E1 +46.501,E3 +158113.137,E4 +0.000} C_DIS
LIN {X -190.147,Y +401.077,Z +0.000,A +0.000,E1 +46.499,E3 +158128.178,E4 +0.000} C_DIS
LIN {X -190.159,Y +390.929,Z +0.000,A +0.000,E1 +46.494,E3 +158141.144,E4 +0.000} C_DIS
LIN {X -190.174,Y +383.973,Z +0.000,A +0.000,E1 +46.484,E3 +158150.037,E4 +0.000} C_DIS
LIN {X -190.200,Y +373.815,Z +0.000,A +0.000,E1 +46.448,E3 +158163.042,E4 +0.000} C_DIS
LIN {X -190.154,Y +361.003,Z +0.000,A +0.000,E1 +46.303,E3 +158179.536,E4 +0.000} C_DIS
LIN {X -189.772,Y +350.660,Z +0.000,A +0.049,E1 +45.996,E3 +158193.075,E4 +0.000} C_DIS
LIN {X -189.325,Y +346.917,Z +0.000,A +0.243,E1 +45.771,E3 +158198.144,E4 +0.000} C_DIS
LIN {X -188.196,Y +342.754,Z +0.000,A +1.966,E1 +45.249,E3 +158204.152,E4 +0.000} C_DIS
LIN {X -185.199,Y +337.023,Z +0.000,A +6.630,E1 +43.793,E3 +158213.526,E4 +0.000} C_DIS
LIN {X -181.141,Y +331.596,Z +0.000,A +12.274,E1 +41.569,E3 +158224.086,E4 +0.000} C_DIS
LIN {X -176.762,Y +326.804,Z +0.000,A +17.560,E1 +38.898,E3 +158235.510,E4 +0.000} C_DIS
LIN {X -172.184,Y +322.578,Z +0.000,A +19.859,E1 +36.197,E3 +158248.240,E4 +0.000} C_DIS
LIN {X -165.998,Y +317.874,Z +0.000,A +20.000,E1 +32.027,E3 +158267.998,E4 +0.000} C_DIS
LIN {X -160.137,Y +314.334,Z +0.000,A +20.000,E1 +26.368,E3 +158292.367,E4 +0.000} C_DIS
LIN {X -155.624,Y +312.245,Z +0.000,A +20.000,E1 +19.506,E3 +158321.043,E4 +0.000} C_DIS
LIN {X -153.557,Y +311.879,Z +0.000,A +20.000,E1 +11.113,E3 +158356.798,E4 +0.000} C_DIS
LIN {X -155.320,Y +313.348,Z +0.000,A +20.000,E1 +3.401,E3 +158389.982,E4 +0.000} C_DIS
LIN {X -160.005,Y +315.804,Z +0.000,A +20.000,E1 -4.720,E3 +158420.360,E4 +0.000} C_DIS
LIN {X -164.504,Y +318.255,Z +0.000,A +20.000,E1 -10.663,E3 +158439.729,E4 +0.000} C_DIS
LIN {X -170.340,Y +322.684,Z +0.000,A +20.000,E1 -17.457,E3 +158459.761,E4 +0.000} C_DIS
LIN {X -175.568,Y +329.106,Z +0.000,A +20.000,E1 -24.747,E3 +158476.995,E4 +0.000} C_DIS
LIN {X -184.074,Y +340.065,Z +0.000,A +20.000,E1 -33.664,E3 +158499.935,E4 +0.000} C_DIS
LIN {X -190.779,Y +351.388,Z +0.000,A +20.000,E1 -40.083,E3 +158517.713,E4 +0.000} C_DIS
LIN {X -195.254,Y +362.955,Z +0.000,A +20.000,E1 -44.515,E3 +158532.466,E4 +0.000} C_DIS
LIN {X -197.754,Y +374.780,Z +0.000,A +20.000,E1 -47.450,E3 +158545.888,E4 +0.000} C_DIS
LIN {X -198.310,Y +383.215,Z +0.000,A +19.956,E1 -48.698,E3 +158555.012,E4 +0.000} C_DIS
LIN {X -197.912,Y +391.275,Z +0.000,A +18.601,E1 -49.158,E3 +158563.730,E4 +0.000} C_DIS
LIN {X -196.679,Y +398.944,Z +0.000,A +13.989,E1 -48.784,E3 +158572.284,E4 +0.000} C_DIS
LIN {X -194.742,Y +406.288,Z +0.000,A +8.476,E1 -48.001,E3 +158580.967,E4 +0.000} C_DIS
LIN {X -192.748,Y +413.472,Z +0.000,A +3.905,E1 -47.267,E3 +158589.977,E4 +0.000} C_DIS
LIN {X -191.781,Y +419.162,Z +0.000,A +1.739,E1 -46.975,E3 +158597.245,E4 +0.000} C_DIS
LIN {X -190.795,Y +430.646,Z +0.000,A +0.152,E1 -46.707,E3 +158611.906,E4 +0.000} C_DIS
LIN {X -190.395,Y +441.145,Z +0.000,A +0.001,E1 -46.583,E3 +158625.299,E4 +0.000} C_DIS
LIN {X -190.239,Y +451.150,Z +0.000,A -0.000,E1 -46.528,E3 +158638.067,E4 +0.000} C_DIS
LIN {X -190.161,Y +465.026,Z +0.000,A -0.000,E1 -46.506,E3 +158655.782,E4 +0.000} C_DIS
LIN {X -190.142,Y +1057.148,Z +0.000,A -0.000,E1 -46.500,E3 +159411.988,E4 +0.000} C_DIS
LIN {X -190.147,Y +1068.924,Z +0.000,A -0.000,E1 -46.499,E3 +159427.029,E4 +0.000} C_DIS
LIN {X -190.159,Y +1079.072,Z +0.000,A -0.000,E1 -46.493,E3 +159439.994,E4 +0.000} C_DIS
LIN {X -190.174,Y +1086.028,Z +0.000,A -0.000,E1 -46.483,E3 +159448.888,E4 +0.000} C_DIS
LIN {X -190.200,Y +1096.186,Z +0.000,A -0.000,E1 -46.448,E3 +159461.892,E4 +0.000} C_DIS
LIN {X -190.154,Y +1108.998,Z +0.000,A -0.054,E1 -46.295,E3 +159478.387,E4 +0.000} C_DIS
LIN {X -189.772,Y +1119.341,Z +0.000,A -0.752,E1 -45.902,E3 +159491.925,E4 +0.000} C_DIS
LIN {X -189.097,Y +1124.276,Z +0.000,A -2.508,E1 -45.397,E3 +159498.657,E4 +0.000} C_DIS
LIN {X -187.410,Y +1129.069,Z +0.000,A -5.304,E1 -44.585,E3 +159505.830,E4 +0.000} C_DIS
LIN {X -183.899,Y +1134.873,Z +0.000,A -10.372,E1 -42.805,E3 +159515.836,E4 +0.000} C_DIS
LIN {X -179.711,Y +1140.065,Z +0.000,A -15.940,E1 -40.393,E3 +159526.622,E4 +0.000} C_DIS
LIN {X -176.763,Y +1143.197,Z +0.000,A -18.748,E1 -38.674,E3 +159534.360,E4 +0.000} C_DIS
LIN {X -172.185,Y +1147.423,Z +0.000,A -19.971,E1 -36.175,E3 +159547.090,E4 +0.000} C_DIS
LIN {X -165.999,Y +1152.127,Z +0.000,A -20.000,E1 -32.027,E3 +159566.848,E4 +0.000} C_DIS
LIN {X -160.138,Y +1155.667,Z +0.000,A -20.000,E1 -26.368,E3 +159591.218,E4 +0.000} C_DIS
LIN {X -155.625,Y +1157.756,Z +0.000,A -20.000,E1 -19.505,E3 +159619.894,E4 +0.000} C_DIS
LIN {X -153.552,Y +1158.113,Z +0.000,A -20.000,E1 -11.113,E3 +159655.645,E4 +0.000} C_DIS
LIN {X -156.311,Y +1155.540,Z +0.000,A -20.000,E1 -0.839,E3 +159699.005,E4 +0.000} C_DIS
LIN {X -161.281,Y +1151.851,Z +0.000,A -20.000,E1 +7.737,E3 +159728.904,E4 +0.000} C_DIS
LIN {X -167.493,Y +1147.157,Z +0.000,A -20.000,E1 +16.195,E3 +159753.343,E4 +0.000} C_DIS
LIN {X -173.235,Y +1142.221,Z +0.000,A -20.000,E1 +22.930,E3 +159770.645,E4 +0.000} C_DIS
LIN {X -181.123,Y +1133.734,Z +0.000,A -20.000,E1 +30.868,E3 +159791.401,E4 +0.000} C_DIS
LIN {X -189.654,Y +1120.856,Z +0.000,A -20.000,E1 +39.018,E3 +159813.415,E4 +0.000} C_DIS
LIN {X -195.246,Y +1107.046,Z +0.000,A -20.000,E1 +44.515,E3 +159831.317,E4 +0.000} C_DIS
LIN {X -198.051,Y +1092.368,Z +0.000,A -20.000,E1 +47.947,E3 +159847.843,E4 +0.000} C_DIS
LIN {X -198.143,Y +1081.370,Z +0.000,A -19.806,E1 +49.153,E3 +159859.704,E4 +0.000} C_DIS
LIN {X -197.177,Y +1073.569,Z +0.000,A -17.356,E1 +49.162,E3 +159868.288,E4 +0.000} C_DIS
LIN {X -195.448,Y +1066.139,Z +0.000,A -12.154,E1 +48.512,E3 +159876.883,E4 +0.000} C_DIS
LIN {X -193.346,Y +1058.941,Z +0.000,A -7.133,E1 +47.724,E3 +159885.763,E4 +0.000} C_DIS
LIN {X -191.781,Y +1050.839,Z +0.000,A -3.715,E1 +47.274,E3 +159896.096,E4 +0.000} C_DIS
LIN {X -190.795,Y +1039.355,Z +0.000,A -0.983,E1 +46.842,E3 +159910.756,E4 +0.000} C_DIS
LIN {X -190.395,Y +1028.856,Z +0.000,A -0.089,E1 +46.598,E3 +159924.150,E4 +0.000} C_DIS
LIN {X -190.239,Y +1018.851,Z +0.000,A -0.004,E1 +46.529,E3 +159936.918,E4 +0.000} C_DIS
LIN {X -190.161,Y +1004.975,Z +0.000,A +0.000,E1 +46.506,E3 +159954.632,E4 +0.000} C_DIS
LIN {X -190.142,Y +412.853,Z +0.000,A +0.000,E1 +46.501,E3 +160710.838,E4 +0.000} C_DIS
LIN {X -190.147,Y +401.077,Z +0.000,A +0.000,E1 +46.499,E3 +160725.879,E4 +0.000} C_DIS
LIN {X -190.159,Y +390.929,Z +0.000,A +0.000,E1 +46.494,E3 +160738.845,E4 +0.000} C_DIS
LIN {X -190.174,Y +383.973,Z +0.000,A +0.000,E1 +46.484,E3 +160747.738,E4 +0.000} C_DIS
LIN {X -190.200,Y +373.815,Z +0.000,A +0.000,E1 +46.448,E3 +160760.743,E4 +0.000} C_DIS
LIN {X -190.154,Y +361.003,Z +0.000,A +0.000,E1 +46.303,E3 +160777.237,E4 +0.000} C_DIS
LIN {X -189.772,Y +350.660,Z +0.000,A +0.049,E1 +45.996,E3 +160790.776,E4 +0.000} C_DIS
LIN {X -189.325,Y +346.917,Z +0.000,A +0.243,E1 +45.771,E3 +160795.845,E4 +0.000} C_DIS
LIN {X -188.196,Y +342.754,Z +0.000,A +1.966,E1 +45.249,E3 +160801.853,E4 +0.000} C_DIS
LIN {X -185.199,Y +337.023,Z +0.000,A +6.630,E1 +43.793,E3 +160811.227,E4 +0.000} C_DIS
LIN {X -181.141,Y +331.596,Z +0.000,A +12.274,E1 +41.569,E3 +160821.787,E4 +0.000} C_DIS
LIN {X -176.762,Y +326.804,Z +0.000,A +17.560,E1 +38.898,E3 +160833.211,E4 +0.000} C_DIS
LIN {X -172.184,Y +322.578,Z +0.000,A +19.859,E1 +36.197,E3 +160845.941,E4 +0.000} C_DIS
LIN {X -165.998,Y +317.874,Z +0.000,A +20.000,E1 +32.027,E3 +160865.699,E4 +0.000} C_DIS
LIN {X -160.137,Y +314.334,Z +0.000,A +20.000,E1 +26.368,E3 +160890.068,E4 +0.000} C_DIS
LIN {X -155.624,Y +312.245,Z +0.000,A +20.000,E1 +19.506,E3 +160918.744,E4 +0.000} C_DIS
LIN {X -153.557,Y +311.879,Z +0.000,A +20.000,E1 +11.113,E3 +160954.499,E4 +0.000} C_DIS
LIN {X -155.320,Y +313.348,Z +0.000,A +20.000,E1 +3.401,E3 +160987.683,E4 +0.000} C_DIS
LIN {X -160.005,Y +315.804,Z +0.000,A +20.000,E1 -4.720,E3 +161018.061,E4 +0.000} C_DIS
LIN {X -164.504,Y +318.255,Z +0.000,A +20.000,E1 -10.663,E3 +161037.430,E4 +0.000} C_DIS
LIN {X -170.340,Y +322.684,Z +0.000,A +20.000,E1 -17.457,E3 +161057.462,E4 +0.000} C_DIS
LIN {X -175.568,Y +329.106,Z +0.000,A +20.000,E1 -24.747,E3 +161074.696,E4 +0.000} C_DIS
LIN {X -184.074,Y +340.065,Z +0.000,A +20.000,E1 -33.664,E3 +161097.636,E4 +0.000} C_DIS
LIN {X -190.779,Y +351.388,Z +0.000,A +20.000,E1 -40.083,E3 +161115.414,E4 +0.000} C_DIS
LIN {X -195.254,Y +362.955,Z +0.000,A +20.000,E1 -44.515,E3 +161130.167,E4 +0.000} C_DIS
LIN {X -197.754,Y +374.780,Z +0.000,A +20.000,E1 -47.450,E3 +161143.589,E4 +0.000} C_DIS
LIN {X -198.310,Y +383.215,Z +0.000,A +19.956,E1 -48.698,E3 +161152.713,E4 +0.000} C_DIS
LIN {X -197.912,Y +391.275,Z +0.000,A +18.601,E1 -49.158,E3 +161161.431,E4 +0.000} C_DIS
LIN {X -196.679,Y +398.944,Z +0.000,A +13.989,E1 -48.784,E3 +161169.985,E4 +0.000} C_DIS
LIN {X -194.742,Y +406.288,Z +0.000,A +8.476,E1 -48.001,E3 +161178.668,E4 +0.000} C_DIS
LIN {X -192.748,Y +413.472,Z +0.000,A +3.905,E1 -47.267,E3 +161187.678,E4 +0.000} C_DIS
LIN {X -191.781,Y +419.162,Z +0.000,A +1.739,E1 -46.975,E3 +161194.946,E4 +0.000} C_DIS
LIN {X -190.795,Y +430.646,Z +0.000,A +0.152,E1 -46.707,E3 +161209.607,E4 +0.000} C_DIS
LIN {X -190.395,Y +441.145,Z +0.000,A +0.001,E1 -46.583,E3 +161223.000,E4 +0.000} C_DIS
LIN {X -190.239,Y +451.150,Z +0.000,A -0.000,E1 -46.528,E3 +161235.768,E4 +0.000} C_DIS
LIN {X -190.161,Y +465.026,Z +0.000,A -0.000,E1 -46.506,E3 +161253.483,E4 +0.000} C_DIS
LIN {X -190.142,Y +1057.148,Z +0.000,A -0.000,E1 -46.500,E3 +162009.689,E4 +0.000} C_DIS
LIN {X -190.147,Y +1068.924,Z +0.000,A -0.000,E1 -46.499,E3 +162024.730,E4 +0.000} C_DIS
LIN {X -190.159,Y +1079.072,Z +0.000,A -0.000,E1 -46.493,E3 +162037.695,E4 +0.000} C_DIS
LIN {X -190.174,Y +1086.028,Z +0.000,A -0.000,E1 -46.483,E3 +162046.589,E4 +0.000} C_DIS
LIN {X -190.200,Y +1096.186,Z +0.000,A -0.000,E1 -46.448,E3 +162059.593,E4 +0.000} C_DIS
LIN {X -190.154,Y +1108.998,Z +0.000,A -0.054,E1 -46.295,E3 +162076.088,E4 +0.000} C_DIS
LIN {X -189.772,Y +1119.341,Z +0.000,A -0.752,E1 -45.902,E3 +162089.626,E4 +0.000} C_DIS
LIN {X -189.097,Y +1124.276,Z +0.000,A -2.508,E1 -45.397,E3 +162096.358,E4 +0.000} C_DIS
LIN {X -187.410,Y +1129.069,Z +0.000,A -5.304,E1 -44.585,E3 +162103.531,E4 +0.000} C_DIS
LIN {X -183.899,Y +1134.873,Z +0.000,A -10.372,E1 -42.805,E3 +162113.537,E4 +0.000} C_DIS
LIN {X -179.711,Y +1140.065,Z +0.000,A -15.940,E1 -40.393,E3 +162124.323,E4 +0.000} C_DIS
LIN {X -176.763,Y +1143.197,Z +0.000,A -18.748,E1 -38.674,E3 +162132.061,E4 +0.000} C_DIS
LIN {X -172.185,Y +1147.423,Z +0.000,A -19.971,E1 -36.175,E3 +162144.791,E4 +0.000} C_DIS
LIN {X -165.999,Y +1152.127,Z +0.000,A -20.000,E1 -32.027,E3 +162164.549,E4 +0.000} C_DIS
LIN {X -160.138,Y +1155.667,Z +0.000,A -20.000,E1 -26.368,E3 +162188.919,E4 +0.000} C_DIS
LIN {X -155.625,Y +1157.756,Z +0.000,A -20.000,E1 -19.505,E3 +162217.595,E4 +0.000} C_DIS
LIN {X -153.552,Y +1158.113,Z +0.000,A -20.000,E1 -11.113,E3 +162253.346,E4 +0.000} C_DIS
LIN {X -156.311,Y +1155.540,Z +0.000,A -20.000,E1 -0.839,E3 +162296.706,E4 +0.000} C_DIS
LIN {X -161.281,Y +1151.851,Z +0.000,A -20.000,E1 +7.737,E3 +162326.605,E4 +0.000} C_DIS
LIN {X -167.493,Y +1147.157,Z +0.000,A -20.000,E1 +16.195,E3 +162351.044,E4 +0.000} C_DIS
LIN {X -173.235,Y +1142.221,Z +0.000,A -20.000,E1 +22.930,E3 +162368.346,E4 +0.000} C_DIS
LIN {X -181.123,Y +1133.734,Z +0.000,A -20.000,E1 +30.868,E3 +162389.102,E4 +0.000} C_DIS
LIN {X -189.654,Y +1120.856,Z +0.000,A -20.000,E1 +39.018,E3 +162411.116,E4 +0.000} C_DIS
LIN {X -195.246,Y +1107.046,Z +0.000,A -20.000,E1 +44.515,E3 +162429.018,E4 +0.000} C_DIS
LIN {X -198.051,Y +1092.368,Z +0.000,A -20.000,E1 +47.947,E3 +162445.544,E4 +0.000} C_DIS
LIN {X -198.143,Y +1081.370,Z +0.000,A -19.806,E1 +49.153,E3 +162457.405,E4 +0.000} C_DIS
LIN {X -197.177,Y +1073.569,Z +0.000,A -17.356,E1 +49.162,E3 +162465.989,E4 +0.000} C_DIS
LIN {X -195.448,Y +1066.139,Z +0.000,A -12.154,E1 +48.512,E3 +162474.584,E4 +0.000} C_DIS
LIN {X -193.346,Y +1058.941,Z +0.000,A -7.133,E1 +47.724,E3 +162483.464,E4 +0.000} C_DIS
LIN {X -191.781,Y +1050.839,Z +0.000,A -3.715,E1 +47.274,E3 +162493.797,E4 +0.000} C_DIS
LIN {X -190.795,Y +1039.355,Z +0.000,A -0.983,E1 +46.842,E3 +162508.457,E4 +0.000} C_DIS
LIN {X -190.395,Y +1028.856,Z +0.000,A -0.089,E1 +46.598,E3 +162521.851,E4 +0.000} C_DIS
LIN {X -190.239,Y +1018.851,Z +0.000,A -0.004,E1 +46.529,E3 +162534.619,E4 +0.000} C_DIS
LIN {X -190.161,Y +1004.975,Z +0.000,A +0.000,E1 +46.506,E3 +162552.333,E4 +0.000} C_DIS
LIN {X -190.142,Y +412.853,Z +0.000,A +0.000,E1 +46.501,E3 +163308.539,E4 +0.000} C_DIS
LIN {X -190.147,Y +401.077,Z +0.000,A +0.000,E1 +46.499,E3 +163323.580,E4 +0.000} C_DIS
LIN {X -190.159,Y +390.929,Z +0.000,A +0.000,E1 +46.494,E3 +163336.546,E4 +0.000} C_DIS
LIN {X -190.174,Y +383.973,Z +0.000,A +0.000,E1 +46.484,E3 +163345.439,E4 +0.000} C_DIS
LIN {X -190.200,Y +373.815,Z +0.000,A +0.000,E1 +46.448,E3 +163358.444,E4 +0.000} C_DIS
LIN {X -190.154,Y +361.003,Z +0.000,A +0.000,E1 +46.303,E3 +163374.938,E4 +0.000} C_DIS
LIN {X -189.772,Y +350.660,Z +0.000,A +0.049,E1 +45.996,E3 +163388.477,E4 +0.000} C_DIS
LIN {X -189.325,Y +346.917,Z +0.000,A +0.243,E1 +45.771,E3 +163393.546,E4 +0.000} C_DIS
LIN {X -188.196,Y +342.754,Z +0.000,A +1.966,E1 +45.249,E3 +163399.554,E4 +0.000} C_DIS
LIN {X -185.199,Y +337.023,Z +0.000,A +6.630,E1 +43.793,E3 +163408.928,E4 +0.000} C_DIS
LIN {X -181.141,Y +331.596,Z +0.000,A +12.274,E1 +41.569,E3 +163419.488,E4 +0.000} C_DIS
LIN {X -176.762,Y +326.804,Z +0.000,A +17.560,E1 +38.898,E3 +163430.912,E4 +0.000} C_DIS
LIN {X -172.184,Y +322.578,Z +0.000,A +19.859,E1 +36.197,E3 +163443.642,E4 +0.000} C_DIS
LIN {X -165.998,Y +317.874,Z +0.000,A +20.000,E1 +32.027,E3 +163463.400,E4 +0.000} C_DIS
LIN {X -160.137,Y +314.334,Z +0.000,A +20.000,E1 +26.368,E3 +163487.769,E4 +0.000} C_DIS
LIN {X -155.624,Y +312.245,Z +0.000,A +20.000,E1 +19.506,E3 +163516.445,E4 +0.000} C_DIS
LIN {X -153.557,Y +311.879,Z +0.000,A +20.000,E1 +11.113,E3 +163552.200,E4 +0.000} C_DIS
LIN {X -155.320,Y +313.348,Z +0.000,A +20.000,E1 +3.401,E3 +163585.384,E4 +0.000} C_DIS
LIN {X -160.005,Y +315.804,Z +0.000,A +20.000,E1 -4.720,E3 +163615.762,E4 +0.000} C_DIS
LIN {X -164.504,Y +318.255,Z +0.000,A +20.000,E1 -10.663,E3 +163635.131,E4 +0.000} C_DIS
LIN {X -170.340,Y +322.684,Z +0.000,A +20.000,E1 -17.457,E3 +163655.163,E4 +0.000} C_DIS
LIN {X -175.568,Y +329.106,Z +0.000,A +20.000,E1 -24.747,E3 +163672.397,E4 +0.000} C_DIS
LIN {X -184.074,Y +340.065,Z +0.000,A +20.000,E1 -33.664,E3 +163695.337,E4 +0.000} C_DIS
LIN {X -190.779,Y +351.388,Z +0.000,A +20.000,E1 -40.083,E3 +163713.115,E4 +0.000} C_DIS
LIN {X -195.254,Y +362.955,Z +0.000,A +20.000,E1 -44.515,E3 +163727.868,E4 +0.000} C_DIS
LIN {X -197.754,Y +374.780,Z +0.000,A +20.000,E1 -47.450,E3 +163741.290,E4 +0.000} C_DIS
LIN {X -198.310,Y +383.215,Z +0.000,A +19.956,E1 -48.698,E3 +163750.414,E4 +0.000} C_DIS
LIN {X -197.912,Y +391.275,Z +0.000,A +18.601,E1 -49.158,E3 +163759.132,E4 +0.000} C_DIS
LIN {X -196.679,Y +398.944,Z +0.000,A +13.989,E1 -48.784,E3 +163767.686,E4 +0.000} C_DIS
LIN {X -194.742,Y +406.288,Z +0.000,A +8.476,E1 -48.001,E3 +163776.369,E4 +0.000} C_DIS
LIN {X -192.748,Y +413.472,Z +0.000,A +3.905,E1 -47.267,E3 +163785.379,E4 +0.000} C_DIS
LIN {X -191.781,Y +419.162,Z +0.000,A +1.739,E1 -46.975,E3 +163792.647,E4 +0.000} C_DIS
LIN {X -190.795,Y +430.646,Z +0.000,A +0.152,E1 -46.707,E3 +163807.308,E4 +0.000} C_DIS
LIN {X -190.395,Y +441.145,Z +0.000,A +0.001,E1 -46.583,E3 +163820.701,E4 +0.000} C_DIS
LIN {X -190.239,Y +451.150,Z +0.000,A -0.000,E1 -46.528,E3 +163833.469,E4 +0.000} C_DIS
LIN {X -190.161,Y +465.026,Z +0.000,A -0.000,E1 -46.506,E3 +163851.184,E4 +0.000} C_DIS
LIN {X -190.142,Y +1057.148,Z +0.000,A -0.000,E1 -46.500,E3 +164607.390,E4 +0.000} C_DIS
LIN {X -190.147,Y +1068.924,Z +0.000,A -0.000,E1 -46.499,E3 +164622.431,E4 +0.000} C_DIS
LIN {X -190.159,Y +1079.072,Z +0.000,A -0.000,E1 -46.493,E3 +164635.396,E4 +0.000} C_DIS
LIN {X -190.174,Y +1086.028,Z +0.000,A -0.000,E1 -46.483,E3 +164644.290,E4 +0.000} C_DIS
LIN {X -190.200,Y +1096.186,Z +0.000,A -0.000,E1 -46.448,E3 +164657.294,E4 +0.000} C_DIS
LIN {X -190.154,Y +1108.998,Z +0.000,A -0.054,E1 -46.295,E3 +164673.789,E4 +0.000} C_DIS
LIN {X -189.772,Y +1119.341,Z +0.000,A -0.752,E1 -45.902,E3 +164687.327,E4 +0.000} C_DIS
LIN {X -189.097,Y +1124.276,Z +0.000,A -2.508,E1 -45.397,E3 +164694.059,E4 +0.000} C_DIS
LIN {X -187.410,Y +1129.069,Z +0.000,A -5.304,E1 -44.585,E3 +164701.232,E4 +0.000} C_DIS
LIN {X -183.899,Y +1134.873,Z +0.000,A -10.372,E1 -42.805,E3 +164711.238,E4 +0.000} C_DIS
LIN {X -179.711,Y +1140.065,Z +0.000,A -15.940,E1 -40.393,E3 +164722.024,E4 +0.000} C_DIS
LIN {X -176.763,Y +1143.197,Z +0.000,A -18.748,E1 -38.674,E3 +164729.762,E4 +0.000} C_DIS
LIN {X -172.185,Y +1147.423,Z +0.000,A -19.971,E1 -36.175,E3 +164742.492,E4 +0.000} C_DIS
LIN {X -165.999,Y +1152.127,Z +0.000,A -20.000,E1 -32.027,E3 +164762.250,E4 +0.000} C_DIS
LIN {X -160.138,Y +1155.667,Z +0.000,A -20.000,E1 -26.368,E3 +164786.620,E4 +0.000} C_DIS
LIN {X -155.625,Y +1157.756,Z +0.000,A -20.000,E1 -19.505,E3 +164815.296,E4 +0.000} C_DIS
LIN {X -153.552,Y +1158.113,Z +0.000,A -20.000,E1 -11.113,E3 +164851.047,E4 +0.000} C_DIS
LIN {X -156.311,Y +1155.540,Z +0.000,A -20.000,E1 -0.839,E3 +164894.407,E4 +0.000} C_DIS
LIN {X -161.281,Y +1151.851,Z +0.000,A -20.000,E1 +7.737,E3 +164924.306,E4 +0.000} C_DIS
LIN {X -167.493,Y +1147.157,Z +0.000,A -20.000,E1 +16.195,E3 +164948.745,E4 +0.000} C_DIS
LIN {X -173.235,Y +1142.221,Z +0.000,A -20.000,E1 +22.930,E3 +164966.047,E4 +0.000} C_DIS
LIN {X -181.123,Y +1133.734,Z +0.000,A -20.000,E1 +30.868,E3 +164986.803,E4 +0.000} C_DIS
LIN {X -189.654,Y +1120.856,Z +0.000,A -20.000,E1 +39.018,E3 +165008.817,E4 +0.000} C_DIS
LIN {X -195.246,Y +1107.046,Z +0.000,A -20.000,E1 +44.515,E3 +165026.719,E4 +0.000} C_DIS
LIN {X -198.051,Y +1092.368,Z +0.000,A -20.000,E1 +47.947,E3 +165043.245,E4 +0.000} C_DIS
LIN {X -198.143,Y +1081.370,Z +0.000,A -19.806,E1 +49.153,E3 +165055.106,E4 +0.000} C_DIS
LIN {X -197.177,Y +1073.569,Z +0.000,A -17.356,E1 +49.162,E3 +165063.690,E4 +0.000} C_DIS
LIN {X -195.448,Y +1066.139,Z +0.000,A -12.154,E1 +48.512,E3 +165072.285,E4 +0.000} C_DIS
LIN {X -193.346,Y +1058.941,Z +0.000,A -7.133,E1 +47.724,E3 +165081.165,E4 +0.000} C_DIS
LIN {X -191.781,Y +1050.839,Z +0.000,A -3.715,E1 +47.274,E3 +165091.498,E4 +0.000} C_DIS
LIN {X -190.795,Y +1039.355,Z +0.000,A -0.983,E1 +46.842,E3 +165106.158,E4 +0.000} C_DIS
LIN {X -190.395,Y +1028.856,Z +0.000,A -0.089,E1 +46.598,E3 +165119.552,E4 +0.000} C_DIS
LIN {X -190.239,Y +1018.851,Z +0.000,A -0.004,E1 +46.529,E3 +165132.320,E4 +0.000} C_DIS
LIN {X -190.161,Y +1004.975,Z +0.000,A +0.000,E1 +46.506,E3 +165150.034,E4 +0.000} C_DIS
LIN {X -190.142,Y +412.853,Z +0.000,A +0.000,E1 +46.501,E3 +165906.240,E4 +0.000} C_DIS
LIN {X -190.147,Y +401.077,Z +0.000,A +0.000,E1 +46.499,E3 +165921.281,E4 +0.000} C_DIS
LIN {X -190.159,Y +390.929,Z +0.000,A +0.000,E1 +46.494,E3 +165934.247,E4 +0.000} C_DIS
LIN {X -190.174,Y +383.973,Z +0.000,A +0.000,E1 +46.484,E3 +165943.140,E4 +0.000} C_DIS
LIN {X -190.200,Y +373.815,Z +0.000,A +0.000,E1 +46.448,E3 +165956.145,E4 +0.000} C_DIS
LIN {X -190.154,Y +361.003,Z +0.000,A +0.000,E1 +46.303,E3 +165972.639,E4 +0.000} C_DIS
LIN {X -189.772,Y +350.660,Z +0.000,A +0.049,E1 +45.996,E3 +165986.178,E4 +0.000} C_DIS
LIN {X -189.325,Y +346.917,Z +0.000,A +0.243,E1 +45.771,E3 +165991.247,E4 +0.000} C_DIS
LIN {X -188.196,Y +342.754,Z +0.000,A +1.966,E1 +45.249,E3 +165997.255,E4 +0.000} C_DIS
LIN {X -185.199,Y +337.023,Z +0.000,A +6.630,E1 +43.793,E3 +166006.629,E4 +0.000} C_DIS
LIN {X -181.141,Y +331.596,Z +0.000,A +12.274,E1 +41.569,E3 +166017.189,E4 +0.000} C_DIS
LIN {X -176.762,Y +326.804,Z +0.000,A +17.560,E1 +38.898,E3 +166028.613,E4 +0.000} C_DIS
LIN {X -172.184,Y +322.578,Z +0.000,A +19.859,E1 +36.197,E3 +166041.343,E4 +0.000} C_DIS
LIN {X -165.998,Y +317.874,Z +0.000,A +20.000,E1 +32.027,E3 +166061.101,E4 +0.000} C_DIS
LIN {X -160.137,Y +314.334,Z +0.000,A +20.000,E1 +26.368,E3 +166085.470,E4 +0.000} C_DIS
LIN {X -155.624,Y +312.245,Z +0.000,A +20.000,E1 +19.506,E3 +166114.146,E4 +0.000} C_DIS
LIN {X -153.557,Y +311.879,Z +0.000,A +20.000,E1 +11.113,E3 +166149.901,E4 +0.000} C_DIS
LIN {X -155.320,Y +313.348,Z +0.000,A +20.000,E1 +3.401,E3 +166183.085,E4 +0.000} C_DIS
LIN {X -160.005,Y +315.804,Z +0.000,A +20.000,E1 -4.720,E3 +166213.463,E4 +0.000} C_DIS
LIN {X -164.504,Y +318.255,Z +0.000,A +20.000,E1 -10.663,E3 +166232.832,E4 +0.000} C_DIS
LIN {X -170.340,Y +322.684,Z +0.000,A +20.000,E1 -17.457,E3 +166252.864,E4 +0.000} C_DIS
LIN {X -175.568,Y +329.106,Z +0.000,A +20.000,E1 -24.747,E3 +166270.098,E4 +0.000} C_DIS
LIN {X -184.074,Y +340.065,Z +0.000,A +20.000,E1 -33.664,E3 +166293.038,E4 +0.000} C_DIS
LIN {X -190.779,Y +351.388,Z +0.000,A +20.000,E1 -40.083,E3 +166310.816,E4 +0.000} C_DIS
LIN {X -195.254,Y +362.955,Z +0.000,A +20.000,E1 -44.515,E3 +166325.569,E4 +0.000} C_DIS
LIN {X -197.754,Y +374.780,Z +0.000,A +20.000,E1 -47.450,E3 +166338.991,E4 +0.000} C_DIS
LIN {X -198.310,Y +383.215,Z +0.000,A +19.956,E1 -48.698,E3 +166348.115,E4 +0.000} C_DIS
LIN {X -197.912,Y +391.275,Z +0.000,A +18.601,E1 -49.158,E3 +166356.833,E4 +0.000} C_DIS
LIN {X -196.679,Y +398.944,Z +0.000,A +13.989,E1 -48.784,E3 +166365.387,E4 +0.000} C_DIS
LIN {X -194.742,Y +406.288,Z +0.000,A +8.476,E1 -48.001,E3 +166374.070,E4 +0.000} C_DIS
LIN {X -192.748,Y +413.472,Z +0.000,A +3.905,E1 -47.267,E3 +166383.080,E4 +0.000} C_DIS
LIN {X -191.781,Y +419.162,Z +0.000,A +1.739,E1 -46.975,E3 +166390.348,E4 +0.000} C_DIS
LIN {X -190.795,Y +430.646,Z +0.000,A +0.152,E1 -46.707,E3 +166405.009,E4 +0.000} C_DIS
LIN {X -190.395,Y +441.145,Z +0.000,A +0.001,E1 -46.583,E3 +166418.402,E4 +0.000} C_DIS
LIN {X -190.239,Y +451.150,Z +0.000,A -0.000,E1 -46.528,E3 +166431.170,E4 +0.000} C_DIS
LIN {X -190.161,Y +465.026,Z +0.000,A -0.000,E1 -46.506,E3 +166448.885,E4 +0.000} C_DIS
LIN {X -190.142,Y +1057.148,Z +0.000,A -0.000,E1 -46.500,E3 +167205.091,E4 +0.000} C_DIS
LIN {X -190.147,Y +1068.924,Z +0.000,A -0.000,E1 -46.499,E3 +167220.132,E4 +0.000} C_DIS
LIN {X -190.159,Y +1079.072,Z +0.000,A -0.000,E1 -46.493,E3 +167233.097,E4 +0.000} C_DIS
LIN {X -190.174,Y +1086.028,Z +0.000,A -0.000,E1 -46.483,E3 +167241.991,E4 +0.000} C_DIS
LIN {X -190.200,Y +1096.186,Z +0.000,A -0.000,E1 -46.448,E3 +167254.995,E4 +0.000} C_DIS
LIN {X -190.154,Y +1108.998,Z +0.000,A -0.054,E1 -46.295,E3 +167271.490,E4 +0.000} C_DIS
LIN {X -189.772,Y +1119.341,Z +0.000,A -0.752,E1 -45.902,E3 +167285.028,E4 +0.000} C_DIS
LIN {X -189.097,Y +1124.276,Z +0.000,A -2.508,E1 -45.397,E3 +167291.760,E4 +0.000} C_DIS
LIN {X -187.410,Y +1129.069,Z +0.000,A -5.304,E1 -44.585,E3 +167298.933,E4 +0.000} C_DIS
LIN {X -183.899,Y +1134.873,Z +0.000,A -10.372,E1 -42.805,E3 +167308.939,E4 +0.000} C_DIS
LIN {X -179.711,Y +1140.065,Z +0.000,A -15.940,E1 -40.393,E3 +167319.725,E4 +0.000} C_DIS
LIN {X -176.763,Y +1143.197,Z +0.000,A -18.748,E1 -38.674,E3 +167327.463,E4 +0.000} C_DIS
LIN {X -172.185,Y +1147.423,Z +0.000,A -19.971,E1 -36.175,E3 +167340.193,E4 +0.000} C_DIS
LIN {X -165.999,Y +1152.127,Z +0.000,A -20.000,E1 -32.027,E3 +167359.951,E4 +0.000} C_DIS
LIN {X -160.138,Y +1155.667,Z +0.000,A -20.000,E1 -26.368,E3 +167384.321,E4 +0.000} C_DIS
LIN {X -155.625,Y +1157.756,Z +0.000,A -20.000,E1 -19.505,E3 +167412.997,E4 +0.000} C_DIS
LIN {X -153.552,Y +1158.113,Z +0.000,A -20.000,E1 -11.113,E3 +167448.748,E4 +0.000} C_DIS
LIN {X -156.311,Y +1155.540,Z +0.000,A -20.000,E1 -0.839,E3 +167492.108,E4 +0.000} C_DIS
LIN {X -161.281,Y +1151.851,Z +0.000,A -20.000,E1 +7.737,E3 +167522.007,E4 +0.000} C_DIS
LIN {X -167.493,Y +1147.157,Z +0.000,A -20.000,E1 +16.195,E3 +167546.446,E4 +0.000} C_DIS
LIN {X -173.235,Y +1142.221,Z +0.000,A -20.000,E1 +22.930,E3 +167563.748,E4 +0.000} C_DIS
LIN {X -181.123,Y +1133.734,Z +0.000,A -20.000,E1 +30.868,E3 +167584.504,E4 +0.000} C_DIS
LIN {X -189.654,Y +1120.856,Z +0.000,A -20.000,E1 +39.018,E3 +167606.518,E4 +0.000} C_DIS
